KUKA KRL program: Machining1.src

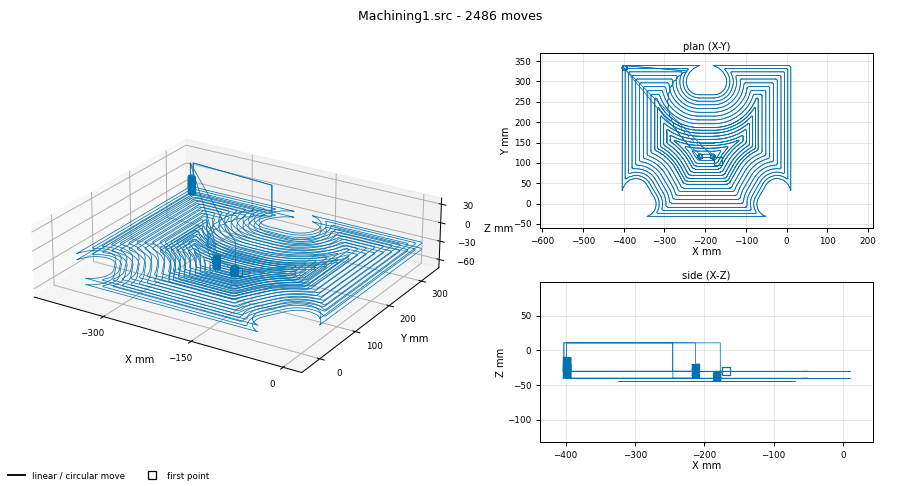
[picture p0: tool path of Machining1.src, 2486 of 2486 moves have a stored position in this frame; points joined in program order, loops and branches not executed]
&ACCESS RVP
&REL 1
&PARAM TEMPLATE = C:\KRC\Roboter\Template\vorgabe
&PARAM EDITMASK = *
DEF Machining1 ( )

; External program calls:
EXT Machining2()

CIRC {X -171.302,Y 100.492,Z -30.000,A 0.015,B 0.000,C 180.000},{X -168.190,Y 103.602,Z -30.000,A 0.015,B 0.000,C 180.000} C_DIS
CIRC {X -167.107,Y 105.546,Z -30.000,A 0.015,B 0.000,C -180.000},{X -166.084,Y 107.524,Z -30.000,A 0.015,B -0.000,C -180.000} C_DIS
CIRC {X -165.062,Y 109.501,Z -30.000,A 0.015,B 0.000,C -180.000},{X -163.978,Y 111.446,Z -30.000,A 0.015,B 0.000,C 180.000} C_DIS
CIRC {X -159.665,Y 118.376,Z -30.000,A 0.015,B 0.000,C 180.000},{X -154.910,Y 125.010,Z -30.000,A 0.015,B -0.000,C -180.000} C_DIS
CIRC {X -149.826,Y 131.393,Z -30.000,A 0.015,B 0.000,C 180.000},{X -144.514,Y 137.587,Z -30.000,A 0.015,B -0.000,C 180.000} C_DIS
CIRC {X -144.313,Y 139.468,Z -30.000,A 0.015,B 0.000,C 180.000},{X -146.029,Y 140.268,Z -30.000,A 0.015,B -0.000,C -180.000} C_DIS
CIRC {X -149.975,Y 139.497,Z -30.000,A 0.015,B 0.000,C -180.000},{X -153.909,Y 138.663,Z -30.000,A 0.015,B 0.000,C 180.000} C_DIS
CIRC {X -157.855,Y 137.887,Z -30.000,A 0.015,B 0.000,C 180.000},{X -161.833,Y 137.294,Z -30.000,A 0.015,B 0.000,C 180.000} C_DIS
CIRC {X -170.208,Y 136.495,Z -30.000,A 0.015,B 0.000,C -180.000},{X -178.617,Y 136.202,Z -30.000,A 0.015,B 0.000,C -180.000} C_DIS
LIN {X -214.895,Y 136.202,Z -30.000,A 0.015,B 0.000,C 180.000} C_DIS
CIRC {X -223.102,Y 136.522,Z -30.000,A 0.015,B 0.000,C 180.000},{X -231.259,Y 137.480,Z -30.000,A 0.015,B 0.000,C 180.000} C_DIS
CIRC {X -232.124,Y 137.616,Z -30.000,A 0.015,B 0.000,C -180.000},{X -232.988,Y 137.754,Z -30.000,A 0.015,B 0.000,C 180.000} C_DIS
CIRC {X -235.696,Y 139.055,Z -30.000,A 0.015,B -0.000,C 180.000},{X -237.254,Y 141.623,Z -30.000,A 0.015,B 0.000,C 180.000} C_DIS
CIRC {X -238.790,Y 144.198,Z -30.000,A 0.015,B 0.000,C 180.000},{X -241.463,Y 145.555,Z -30.000,A 0.015,B 0.000,C 180.000} C_DIS
CIRC {X -243.440,Y 145.946,Z -30.000,A 0.015,B -0.000,C 180.000},{X -245.411,Y 146.366,Z -30.000,A 0.015,B 0.000,C -180.000} C_DIS
CIRC {X -260.252,Y 150.338,Z -30.000,A 0.015,B 0.000,C 180.000},{X -274.679,Y 155.621,Z -30.000,A 0.015,B 0.000,C -180.000} C_DIS
CIRC {X -276.235,Y 155.093,Z -30.000,A 0.015,B -0.000,C -180.000},{X -275.907,Y 153.483,Z -30.000,A 0.015,B 0.000,C -180.000} C_DIS
CIRC {X -266.896,Y 146.130,Z -30.000,A 0.015,B -0.000,C -180.000},{X -258.464,Y 138.119,Z -30.000,A 0.015,B 0.000,C -180.000} C_DIS
CIRC {X -250.617,Y 129.537,Z -30.000,A 0.015,B 0.000,C 180.000},{X -243.351,Y 120.458,Z -30.000,A 0.015,B -0.000,C 180.000} C_DIS
CIRC {X -241.131,Y 117.362,Z -30.000,A 0.015,B 0.000,C -180.000},{X -239.037,Y 114.180,Z -30.000,A 0.015,B 0.000,C 180.000} C_DIS
CIRC {X -237.039,Y 110.937,Z -30.000,A 0.015,B -0.000,C -180.000},{X -235.105,Y 107.656,Z -30.000,A 0.015,B 0.000,C 180.000} C_DIS
CIRC {X -233.604,Y 104.954,Z -30.000,A 0.015,B 0.000,C 180.000},{X -232.188,Y 102.206,Z -30.000,A 0.015,B 0.000,C 180.000} C_DIS
CIRC {X -230.772,Y 99.459,Z -30.000,A 0.015,B 0.000,C -180.000},{X -229.270,Y 96.757,Z -30.000,A 0.015,B 0.000,C -180.000} C_DIS
CIRC {X -226.165,Y 93.648,Z -30.000,A 0.015,B 0.000,C 180.000},{X -221.922,Y 92.510,Z -30.000,A 0.015,B 0.000,C 180.000} C_DIS
LIN {X -171.602,Y 92.510,Z -30.000,A 0.015,B 0.000,C -180.000} C_DIS
CIRC {X -167.353,Y 93.648,Z -30.000,A 0.015,B 0.000,C -180.000},{X -164.241,Y 96.758,Z -30.000,A 0.015,B 0.000,C 180.000} C_DIS
CIRC {X -162.677,Y 99.566,Z -30.000,A 0.015,B 0.000,C 180.000},{X -161.200,Y 102.421,Z -30.000,A 0.015,B -0.000,C 180.000} C_DIS
CIRC {X -159.724,Y 105.276,Z -30.000,A 0.015,B 0.000,C 180.000},{X -158.160,Y 108.083,Z -30.000,A 0.015,B 0.000,C -180.000} C_DIS
CIRC {X -149.792,Y 120.931,Z -30.000,A 0.015,B -0.000,C -180.000},{X -140.107,Y 132.817,Z -30.000,A 0.015,B -0.000,C -180.000} C_DIS
CIRC {X -129.299,Y 143.685,Z -30.000,A 0.015,B 0.000,C -180.000},{X -117.547,Y 153.523,Z -30.000,A 0.015,B -0.000,C 180.000} C_DIS
CIRC {X -117.226,Y 155.134,Z -30.000,A 0.015,B 0.000,C 180.000},{X -118.785,Y 155.652,Z -30.000,A 0.015,B 0.000,C 180.000} C_DIS
CIRC {X -129.422,Y 151.590,Z -30.000,A 0.015,B 0.000,C -180.000},{X -140.331,Y 148.327,Z -30.000,A 0.015,B 0.000,C 180.000} C_DIS
CIRC {X -151.437,Y 145.826,Z -30.000,A 0.015,B -0.000,C -180.000},{X -162.682,Y 144.043,Z -30.000,A 0.015,B 0.000,C 180.000} C_DIS
CIRC {X -170.633,Y 143.295,Z -30.000,A 0.015,B 0.000,C 180.000},{X -178.617,Y 143.045,Z -30.000,A 0.015,B 0.000,C 180.000} C_DIS
LIN {X -214.895,Y 143.045,Z -30.000,A 0.015,B 0.000,C 180.000} C_DIS
CIRC {X -228.238,Y 143.674,Z -30.000,A 0.015,B 0.000,C 180.000},{X -241.463,Y 145.555,Z -30.000,A 0.015,B 0.000,C -180.000} C_DIS
CIRC {X -244.234,Y 147.015,Z -30.000,A 0.015,B 0.000,C 180.000},{X -245.715,Y 149.775,Z -30.000,A 0.015,B 0.000,C -180.000} C_DIS
CIRC {X -247.142,Y 152.546,Z -30.000,A 0.015,B 0.000,C -180.000},{X -249.821,Y 154.137,Z -30.000,A 0.015,B -0.000,C -180.000} C_DIS
LIN {X -250.098,Y 154.210,Z -30.000,A 0.015,B -0.000,C -180.000} C_DIS
CIRC {X -267.011,Y 159.678,Z -30.000,A 0.015,B 0.000,C -180.000},{X -283.228,Y 166.955,Z -30.000,A 0.015,B 0.000,C 180.000} C_DIS
CIRC {X -285.491,Y 166.874,Z -30.000,A 0.015,B 0.000,C -180.000},{X -286.600,Y 164.900,Z -30.000,A 0.015,B 0.000,C 180.000} C_DIS
LIN {X -286.600,Y 156.568,Z -30.000,A 0.015,B 0.000,C 180.000} C_DIS
CIRC {X -285.833,Y 153.428,Z -30.000,A 0.015,B 0.000,C 180.000},{X -283.705,Y 150.996,Z -30.000,A 0.015,B 0.000,C 180.000} C_DIS
CIRC {X -271.141,Y 141.152,Z -30.000,A 0.015,B 0.000,C -180.000},{X -259.666,Y 130.058,Z -30.000,A 0.015,B 0.000,C -180.000} C_DIS
CIRC {X -249.460,Y 117.780,Z -30.000,A 0.015,B 0.000,C 180.000},{X -240.715,Y 104.423,Z -30.000,A 0.015,B 0.000,C -180.000} C_DIS
CIRC {X -238.751,Y 100.888,Z -30.000,A 0.015,B 0.000,C 180.000},{X -236.898,Y 97.293,Z -30.000,A 0.015,B 0.000,C -180.000} C_DIS
CIRC {X -235.045,Y 93.698,Z -30.000,A 0.015,B -0.000,C -180.000},{X -233.081,Y 90.163,Z -30.000,A 0.015,B -0.000,C -180.000} C_DIS
CIRC {X -229.976,Y 87.054,Z -30.000,A 0.015,B 0.000,C 180.000},{X -225.732,Y 85.916,Z -30.000,A 0.015,B 0.000,C 180.000} C_DIS
LIN {X -167.797,Y 85.916,Z -30.000,A 0.015,B 0.000,C 180.000} C_DIS
CIRC {X -163.547,Y 87.055,Z -30.000,A 0.015,B -0.000,C 180.000},{X -160.436,Y 90.164,Z -30.000,A 0.015,B 0.000,C 180.000} C_DIS
CIRC {X -158.408,Y 93.803,Z -30.000,A 0.015,B 0.000,C -180.000},{X -156.495,Y 97.504,Z -30.000,A 0.015,B 0.000,C -180.000} C_DIS
CIRC {X -154.582,Y 101.205,Z -30.000,A 0.015,B 0.000,C 180.000},{X -152.554,Y 104.844,Z -30.000,A 0.015,B 0.000,C -180.000} C_DIS
CIRC {X -143.851,Y 118.092,Z -30.000,A 0.015,B 0.000,C 180.000},{X -133.694,Y 130.260,Z -30.000,A 0.015,B 0.000,C 180.000} C_DIS
CIRC {X -122.283,Y 141.253,Z -30.000,A 0.015,B 0.000,C 180.000},{X -109.806,Y 151.020,Z -30.000,A 0.015,B -0.000,C -180.000} C_DIS
CIRC {X -107.679,Y 153.453,Z -30.000,A 0.015,B 0.000,C 180.000},{X -106.912,Y 156.592,Z -30.000,A 0.015,B 0.000,C -180.000} C_DIS
LIN {X -106.913,Y 164.900,Z -30.000,A 0.015,B -0.000,C 180.000} C_DIS
CIRC {X -108.021,Y 166.866,Z -30.000,A 0.015,B 0.000,C -180.000},{X -110.278,Y 166.935,Z -30.000,A 0.015,B 0.000,C 180.000} C_DIS
CIRC {X -122.965,Y 161.035,Z -30.000,A 0.015,B 0.000,C 180.000},{X -136.157,Y 156.372,Z -30.000,A 0.015,B -0.000,C -180.000} C_DIS
CIRC {X -149.710,Y 152.908,Z -30.000,A 0.015,B -0.000,C -180.000},{X -163.504,Y 150.586,Z -30.000,A 0.015,B -0.000,C -180.000} C_DIS
CIRC {X -171.046,Y 149.876,Z -30.000,A 0.015,B 0.000,C 180.000},{X -178.617,Y 149.639,Z -30.000,A 0.015,B 0.000,C 180.000} C_DIS
LIN {X -214.895,Y 149.639,Z -30.000,A 0.015,B 0.000,C -180.000} C_DIS
CIRC {X -232.503,Y 150.768,Z -30.000,A 0.015,B -0.000,C 180.000},{X -249.821,Y 154.137,Z -30.000,A 0.015,B -0.000,C 180.000} C_DIS
CIRC {X -253.023,Y 156.105,Z -30.000,A 0.015,B 0.000,C -180.000},{X -254.587,Y 159.522,Z -30.000,A 0.015,B 0.000,C -180.000} C_DIS
CIRC {X -256.087,Y 162.948,Z -30.000,A 0.015,B 0.000,C 180.000},{X -259.170,Y 165.064,Z -30.000,A 0.015,B 0.000,C 180.000} C_DIS
CIRC {X -269.017,Y 168.755,Z -30.000,A 0.015,B 0.000,C -180.000},{X -278.578,Y 173.132,Z -30.000,A 0.015,B 0.000,C -180.000} C_DIS
CIRC {X -281.907,Y 174.946,Z -30.000,A 0.015,B 0.000,C -180.000},{X -285.103,Y 176.984,Z -30.000,A 0.015,B 0.000,C 180.000} C_DIS
CIRC {X -288.241,Y 179.109,Z -30.000,A 0.015,B 0.000,C 180.000},{X -291.406,Y 181.191,Z -30.000,A 0.015,B 0.000,C 180.000} C_DIS
CIRC {X -293.577,Y 181.275,Z -30.000,A 0.015,B 0.000,C 180.000},{X -294.687,Y 179.408,Z -30.000,A 0.015,B 0.000,C 180.000} C_DIS
LIN {X -294.686,Y 153.798,Z -30.000,A 0.015,B 0.000,C 180.000} C_DIS
CIRC {X -293.590,Y 149.349,Z -30.000,A 0.015,B 0.000,C 180.000},{X -290.552,Y 145.919,Z -30.000,A 0.015,B 0.000,C 180.000} C_DIS
CIRC {X -271.422,Y 130.249,Z -30.000,A 0.015,B 0.000,C -180.000},{X -255.107,Y 111.666,Z -30.000,A 0.015,B 0.000,C 180.000} C_DIS
CIRC {X -251.230,Y 106.146,Z -30.000,A 0.015,B 0.000,C 180.000},{X -247.689,Y 100.404,Z -30.000,A 0.015,B -0.000,C 180.000} C_DIS
CIRC {X -245.145,Y 95.855,Z -30.000,A 0.015,B -0.000,C 180.000},{X -242.722,Y 91.240,Z -30.000,A 0.015,B 0.000,C 180.000} C_DIS
CIRC {X -240.298,Y 86.626,Z -30.000,A 0.015,B 0.000,C 180.000},{X -237.754,Y 82.077,Z -30.000,A 0.015,B 0.000,C -180.000} C_DIS
CIRC {X -234.649,Y 78.968,Z -30.000,A 0.015,B 0.000,C 180.000},{X -230.405,Y 77.830,Z -30.000,A 0.015,B 0.000,C -180.000} C_DIS
LIN {X -163.130,Y 77.830,Z -30.000,A 0.015,B 0.000,C 180.000} C_DIS
CIRC {X -158.881,Y 78.968,Z -30.000,A 0.015,B -0.000,C 180.000},{X -155.769,Y 82.077,Z -30.000,A 0.015,B 0.000,C 180.000} C_DIS
CIRC {X -153.160,Y 86.728,Z -30.000,A 0.015,B 0.000,C 180.000},{X -150.670,Y 91.443,Z -30.000,A 0.015,B 0.000,C 180.000} C_DIS
CIRC {X -148.181,Y 96.158,Z -30.000,A 0.015,B -0.000,C 180.000},{X -145.572,Y 100.809,Z -30.000,A 0.015,B 0.000,C -180.000} C_DIS
CIRC {X -136.969,Y 113.835,Z -30.000,A 0.015,B 0.000,C 180.000},{X -126.877,Y 125.745,Z -30.000,A 0.015,B -0.000,C -180.000} C_DIS
CIRC {X -115.507,Y 136.435,Z -30.000,A 0.015,B 0.000,C 180.000},{X -103.058,Y 145.845,Z -30.000,A 0.015,B 0.000,C -180.000} C_DIS
CIRC {X -99.949,Y 149.299,Z -30.000,A 0.015,B 0.000,C 180.000},{X -98.826,Y 153.807,Z -30.000,A 0.015,B 0.000,C 180.000} C_DIS
LIN {X -98.826,Y 179.417,Z -30.000,A 0.015,B 0.000,C -180.000} C_DIS
CIRC {X -99.933,Y 181.277,Z -30.000,A 0.015,B -0.000,C -180.000},{X -102.095,Y 181.192,Z -30.000,A 0.015,B 0.000,C -180.000} C_DIS
CIRC {X -110.083,Y 176.279,Z -30.000,A 0.015,B 0.000,C 180.000},{X -118.304,Y 171.770,Z -30.000,A 0.015,B -0.000,C -180.000} C_DIS
CIRC {X -126.806,Y 167.804,Z -30.000,A 0.015,B 0.000,C 180.000},{X -135.601,Y 164.537,Z -30.000,A 0.015,B 0.000,C 180.000} C_DIS
CIRC {X -155.043,Y 159.783,Z -30.000,A 0.015,B -0.000,C -180.000},{X -174.979,Y 158.001,Z -30.000,A 0.015,B 0.000,C 180.000} C_DIS
LIN {X -214.895,Y 157.726,Z -30.000,A 0.015,B -0.000,C -180.000} C_DIS
CIRC {X -231.386,Y 158.726,Z -30.000,A 0.015,B 0.000,C 180.000},{X -247.636,Y 161.713,Z -30.000,A 0.015,B 0.000,C -180.000} C_DIS
CIRC {X -253.437,Y 163.272,Z -30.000,A 0.015,B 0.000,C 180.000},{X -259.170,Y 165.064,Z -30.000,A 0.015,B -0.000,C -180.000} C_DIS
CIRC {X -262.205,Y 167.235,Z -30.000,A 0.015,B 0.000,C 180.000},{X -263.500,Y 170.734,Z -30.000,A 0.015,B 0.000,C -180.000} C_DIS
CIRC {X -264.716,Y 174.238,Z -30.000,A 0.015,B 0.000,C 180.000},{X -267.594,Y 176.578,Z -30.000,A 0.015,B -0.000,C 180.000} C_DIS
CIRC {X -271.373,Y 178.266,Z -30.000,A 0.015,B 0.000,C 180.000},{X -275.101,Y 180.067,Z -30.000,A 0.015,B 0.000,C 180.000} C_DIS
CIRC {X -281.532,Y 183.634,Z -30.000,A 0.015,B 0.000,C -180.000},{X -287.644,Y 187.725,Z -30.000,A 0.015,B 0.000,C 180.000} C_DIS
CIRC {X -293.535,Y 192.117,Z -30.000,A 0.015,B -0.000,C -180.000},{X -299.344,Y 196.618,Z -30.000,A 0.015,B 0.000,C -180.000} C_DIS
CIRC {X -301.411,Y 196.843,Z -30.000,A 0.015,B -0.000,C 180.000},{X -302.515,Y 195.081,Z -30.000,A 0.015,B 0.000,C 180.000} C_DIS
LIN {X -302.514,Y 149.210,Z -30.000,A 0.015,B 0.000,C -180.000} C_DIS
CIRC {X -301.418,Y 144.941,Z -30.000,A 0.015,B 0.000,C -180.000},{X -298.400,Y 141.729,Z -30.000,A 0.015,B 0.000,C 180.000} C_DIS
CIRC {X -287.970,Y 134.375,Z -30.000,A 0.015,B 0.000,C 180.000},{X -278.306,Y 126.039,Z -30.000,A 0.015,B 0.000,C 180.000} C_DIS
CIRC {X -269.440,Y 116.864,Z -30.000,A 0.015,B 0.000,C -180.000},{X -261.376,Y 106.977,Z -30.000,A 0.015,B 0.000,C 180.000} C_DIS
CIRC {X -257.767,Y 101.839,Z -30.000,A 0.015,B 0.000,C 180.000},{X -254.471,Y 96.496,Z -30.000,A 0.015,B 0.000,C 180.000} C_DIS
CIRC {X -251.364,Y 90.966,Z -30.000,A 0.015,B -0.000,C -180.000},{X -248.375,Y 85.372,Z -30.000,A 0.015,B -0.000,C 180.000} C_DIS
CIRC {X -245.386,Y 79.778,Z -30.000,A 0.015,B 0.000,C -180.000},{X -242.278,Y 74.249,Z -30.000,A 0.015,B -0.000,C -180.000} C_DIS
CIRC {X -239.173,Y 71.140,Z -30.000,A 0.015,B 0.000,C 180.000},{X -234.929,Y 70.002,Z -30.000,A 0.015,B 0.000,C 180.000} C_DIS
LIN {X -158.613,Y 70.002,Z -30.000,A 0.015,B 0.000,C 180.000} C_DIS
CIRC {X -154.364,Y 71.140,Z -30.000,A 0.015,B 0.000,C 180.000},{X -151.252,Y 74.249,Z -30.000,A 0.015,B 0.000,C -180.000} C_DIS
LIN {X -138.794,Y 96.892,Z -30.000,A 0.015,B 0.000,C -180.000} C_DIS
CIRC {X -130.024,Y 110.028,Z -30.000,A 0.015,B 0.000,C 180.000},{X -119.634,Y 121.923,Z -30.000,A 0.015,B 0.000,C -180.000} C_DIS
CIRC {X -107.912,Y 132.494,Z -30.000,A 0.015,B -0.000,C 180.000},{X -95.112,Y 141.730,Z -30.000,A 0.015,B 0.000,C 180.000} C_DIS
CIRC {X -92.093,Y 144.970,Z -30.000,A 0.015,B 0.000,C 180.000},{X -90.997,Y 149.261,Z -30.000,A 0.015,B 0.000,C -180.000} C_DIS
LIN {X -90.999,Y 195.079,Z -30.000,A 0.015,B 0.000,C 180.000} C_DIS
CIRC {X -92.103,Y 196.841,Z -30.000,A 0.015,B -0.000,C 180.000},{X -94.171,Y 196.616,Z -30.000,A 0.015,B 0.000,C -180.000} C_DIS
CIRC {X -104.346,Y 189.131,Z -30.000,A 0.015,B 0.000,C 180.000},{X -115.009,Y 182.357,Z -30.000,A 0.015,B 0.000,C -180.000} C_DIS
CIRC {X -126.237,Y 176.544,Z -30.000,A 0.015,B -0.000,C 180.000},{X -138.028,Y 171.980,Z -30.000,A 0.015,B 0.000,C -180.000} C_DIS
CIRC {X -156.878,Y 167.393,Z -30.000,A 0.015,B 0.000,C -180.000},{X -176.208,Y 165.732,Z -30.000,A 0.015,B 0.000,C 180.000} C_DIS
LIN {X -214.895,Y 165.554,Z -30.000,A 0.015,B 0.000,C 180.000} C_DIS
CIRC {X -230.483,Y 166.493,Z -30.000,A 0.015,B 0.000,C 180.000},{X -245.845,Y 169.297,Z -30.000,A 0.015,B 0.000,C -180.000} C_DIS
CIRC {X -256.869,Y 172.489,Z -30.000,A 0.015,B -0.000,C 180.000},{X -267.594,Y 176.578,Z -30.000,A 0.015,B 0.000,C 180.000} C_DIS
CIRC {X -270.381,Y 178.951,Z -30.000,A 0.015,B 0.000,C 180.000},{X -271.340,Y 182.484,Z -30.000,A 0.015,B 0.000,C 180.000} C_DIS
CIRC {X -272.205,Y 186.013,Z -30.000,A 0.015,B 0.000,C 180.000},{X -274.787,Y 188.568,Z -30.000,A 0.015,B -0.000,C -180.000} C_DIS
CIRC {X -292.023,Y 200.077,Z -30.000,A 0.015,B -0.000,C -180.000},{X -307.098,Y 214.300,Z -30.000,A 0.015,B 0.000,C 180.000} C_DIS
CIRC {X -308.980,Y 214.762,Z -30.000,A 0.015,B -0.000,C 180.000},{X -310.080,Y 213.167,Z -30.000,A 0.015,B -0.000,C -180.000} C_DIS
LIN {X -310.079,Y 144.563,Z -30.000,A 0.015,B 0.000,C 180.000} C_DIS
CIRC {X -308.981,Y 140.472,Z -30.000,A 0.015,B 0.000,C -180.000},{X -305.984,Y 137.478,Z -30.000,A 0.015,B 0.000,C -180.000} C_DIS
CIRC {X -295.014,Y 130.299,Z -30.000,A 0.015,B 0.000,C 180.000},{X -284.926,Y 121.925,Z -30.000,A 0.015,B -0.000,C -180.000} C_DIS
CIRC {X -275.743,Y 112.578,Z -30.000,A 0.015,B -0.000,C -180.000},{X -267.433,Y 102.447,Z -30.000,A 0.015,B 0.000,C -180.000} C_DIS
CIRC {X -264.084,Y 97.678,Z -30.000,A 0.015,B 0.000,C 180.000},{X -261.025,Y 92.719,Z -30.000,A 0.015,B 0.000,C 180.000} C_DIS
LIN {X -246.650,Y 66.684,Z -30.000,A 0.015,B 0.000,C -180.000} C_DIS
CIRC {X -243.545,Y 63.575,Z -30.000,A 0.015,B 0.000,C -180.000},{X -239.301,Y 62.437,Z -30.000,A 0.015,B 0.000,C 180.000} C_DIS
LIN {X -154.248,Y 62.437,Z -30.000,A 0.015,B 0.000,C -180.000} C_DIS
CIRC {X -149.998,Y 63.575,Z -30.000,A 0.015,B 0.000,C 180.000},{X -146.887,Y 66.685,Z -30.000,A 0.015,B 0.000,C 180.000} C_DIS
LIN {X -132.244,Y 93.107,Z -30.000,A 0.015,B 0.000,C 180.000} C_DIS
CIRC {X -123.362,Y 106.324,Z -30.000,A 0.015,B 0.000,C -180.000},{X -112.778,Y 118.222,Z -30.000,A 0.015,B 0.000,C 180.000} C_DIS
CIRC {X -100.749,Y 128.648,Z -30.000,A 0.015,B 0.000,C -180.000},{X -87.524,Y 137.509,Z -30.000,A 0.015,B 0.000,C -180.000} C_DIS
CIRC {X -84.528,Y 140.526,Z -30.000,A 0.015,B -0.000,C 180.000},{X -83.433,Y 144.635,Z -30.000,A 0.015,B 0.000,C -180.000} C_DIS
LIN {X -83.435,Y 213.163,Z -30.000,A 0.015,B 0.000,C -180.000} C_DIS
CIRC {X -84.535,Y 214.758,Z -30.000,A 0.015,B 0.000,C -180.000},{X -86.417,Y 214.296,Z -30.000,A 0.015,B 0.000,C 180.000} C_DIS
CIRC {X -103.225,Y 198.757,Z -30.000,A 0.015,B 0.000,C -180.000},{X -122.750,Y 186.812,Z -30.000,A 0.015,B 0.000,C 180.000} C_DIS
CIRC {X -144.065,Y 178.566,Z -30.000,A 0.015,B -0.000,C 180.000},{X -166.434,Y 173.881,Z -30.000,A 0.015,B 0.000,C 180.000} C_DIS
LIN {X -214.895,Y 173.118,Z -30.000,A 0.015,B -0.000,C 180.000} C_DIS
CIRC {X -245.822,Y 177.043,Z -30.000,A 0.015,B 0.000,C 180.000},{X -274.787,Y 188.568,Z -30.000,A 0.015,B 0.000,C 180.000} C_DIS
CIRC {X -277.258,Y 191.114,Z -30.000,A 0.015,B 0.000,C 180.000},{X -277.893,Y 194.605,Z -30.000,A 0.015,B 0.000,C -180.000} C_DIS
CIRC {X -278.464,Y 198.089,Z -30.000,A 0.015,B -0.000,C 180.000},{X -280.787,Y 200.746,Z -30.000,A 0.015,B -0.000,C -180.000} C_DIS
CIRC {X -284.969,Y 203.559,Z -30.000,A 0.015,B 0.000,C -180.000},{X -289.045,Y 206.523,Z -30.000,A 0.015,B 0.000,C -180.000} C_DIS
CIRC {X -296.399,Y 212.790,Z -30.000,A 0.015,B 0.000,C -180.000},{X -302.966,Y 219.879,Z -30.000,A 0.015,B 0.000,C 180.000} C_DIS
CIRC {X -308.886,Y 227.498,Z -30.000,A 0.015,B -0.000,C -180.000},{X -314.377,Y 235.434,Z -30.000,A 0.015,B -0.000,C -180.000} C_DIS
CIRC {X -316.098,Y 236.067,Z -30.000,A 0.015,B 0.000,C 180.000},{X -317.194,Y 234.597,Z -30.000,A 0.015,B 0.000,C 180.000} C_DIS
LIN {X -317.192,Y 140.213,Z -30.000,A 0.015,B 0.000,C 180.000} C_DIS
CIRC {X -316.058,Y 136.125,Z -30.000,A 0.015,B 0.000,C -180.000},{X -312.979,Y 133.205,Z -30.000,A 0.015,B 0.000,C -180.000} C_DIS
CIRC {X -292.253,Y 119.088,Z -30.000,A 0.015,B 0.000,C -180.000},{X -275.088,Y 100.805,Z -30.000,A 0.015,B -0.000,C 180.000} C_DIS
CIRC {X -273.004,Y 97.971,Z -30.000,A 0.015,B 0.000,C -180.000},{X -270.965,Y 95.104,Z -30.000,A 0.015,B 0.000,C 180.000} C_DIS
CIRC {X -269.012,Y 92.177,Z -30.000,A 0.015,B 0.000,C 180.000},{X -267.189,Y 89.167,Z -30.000,A 0.015,B 0.000,C 180.000} C_DIS
LIN {X -250.742,Y 59.538,Z -30.000,A 0.015,B 0.000,C 180.000} C_DIS
CIRC {X -247.660,Y 56.453,Z -30.000,A 0.015,B 0.000,C 180.000},{X -243.449,Y 55.324,Z -30.000,A 0.015,B -0.000,C -180.000} C_DIS
LIN {X -150.080,Y 55.324,Z -30.000,A 0.015,B 0.000,C -180.000} C_DIS
CIRC {X -145.885,Y 56.447,Z -30.000,A 0.015,B -0.000,C 180.000},{X -142.813,Y 59.517,Z -30.000,A 0.015,B 0.000,C 180.000} C_DIS
LIN {X -126.086,Y 89.548,Z -30.000,A 0.015,B 0.000,C 180.000} C_DIS
CIRC {X -106.380,Y 114.666,Z -30.000,A 0.015,B 0.000,C -180.000},{X -80.454,Y 133.297,Z -30.000,A 0.015,B 0.000,C -180.000} C_DIS
CIRC {X -77.433,Y 136.144,Z -30.000,A 0.015,B 0.000,C 180.000},{X -76.319,Y 140.143,Z -30.000,A 0.015,B 0.000,C -180.000} C_DIS
LIN {X -76.322,Y 234.602,Z -30.000,A 0.015,B 0.000,C 180.000} C_DIS
CIRC {X -77.419,Y 236.069,Z -30.000,A 0.015,B 0.000,C 180.000},{X -79.136,Y 235.433,Z -30.000,A 0.015,B 0.000,C -180.000} C_DIS
CIRC {X -85.589,Y 226.331,Z -30.000,A 0.015,B 0.000,C -180.000},{X -92.790,Y 217.807,Z -30.000,A 0.015,B -0.000,C 180.000} C_DIS
CIRC {X -100.722,Y 209.957,Z -30.000,A 0.015,B 0.000,C 180.000},{X -109.355,Y 202.884,Z -30.000,A 0.015,B 0.000,C 180.000} C_DIS
CIRC {X -120.709,Y 195.513,Z -30.000,A 0.015,B -0.000,C 180.000},{X -132.910,Y 189.647,Z -30.000,A 0.015,B 0.000,C -180.000} C_DIS
CIRC {X -145.694,Y 185.225,Z -30.000,A 0.015,B 0.000,C 180.000},{X -158.864,Y 182.136,Z -30.000,A 0.015,B -0.000,C -180.000} C_DIS
CIRC {X -172.795,Y 180.330,Z -30.000,A 0.015,B 0.000,C -180.000},{X -186.837,Y 179.928,Z -30.000,A 0.015,B -0.000,C 180.000} C_DIS
LIN {X -214.895,Y 180.232,Z -30.000,A 0.015,B 0.000,C -180.000} C_DIS
CIRC {X -234.824,Y 182.020,Z -30.000,A 0.015,B 0.000,C -180.000},{X -254.115,Y 187.329,Z -30.000,A 0.015,B 0.000,C 180.000} C_DIS
CIRC {X -267.814,Y 193.316,Z -30.000,A 0.015,B 0.000,C -180.000},{X -280.787,Y 200.746,Z -30.000,A 0.015,B 0.000,C 180.000} C_DIS
CIRC {X -282.747,Y 203.101,Z -30.000,A 0.015,B 0.000,C 180.000},{X -283.016,Y 206.154,Z -30.000,A 0.015,B 0.000,C -180.000} C_DIS
CIRC {X -283.201,Y 209.188,Z -30.000,A 0.015,B -0.000,C -180.000},{X -284.951,Y 211.674,Z -30.000,A 0.015,B 0.000,C 180.000} C_DIS
CIRC {X -304.568,Y 232.271,Z -30.000,A 0.015,B 0.000,C 180.000},{X -318.317,Y 257.172,Z -30.000,A 0.015,B 0.000,C -180.000} C_DIS
CIRC {X -321.488,Y 258.916,Z -30.000,A 0.015,B 0.000,C 180.000},{X -323.796,Y 256.128,Z -30.000,A 0.015,B 0.000,C 180.000} C_DIS
LIN {X -323.792,Y 135.950,Z -30.000,A 0.015,B 0.000,C -180.000} C_DIS
CIRC {X -322.699,Y 132.062,Z -30.000,A 0.015,B 0.000,C -180.000},{X -319.740,Y 129.313,Z -30.000,A 0.015,B 0.000,C -180.000} C_DIS
CIRC {X -312.688,Y 125.465,Z -30.000,A 0.015,B 0.000,C 180.000},{X -305.836,Y 121.270,Z -30.000,A 0.015,B 0.000,C 180.000} C_DIS
CIRC {X -299.286,Y 116.609,Z -30.000,A 0.015,B 0.000,C -180.000},{X -293.174,Y 111.386,Z -30.000,A 0.015,B 0.000,C -180.000} C_DIS
CIRC {X -281.197,Y 98.287,Z -30.000,A 0.015,B 0.000,C 180.000},{X -271.423,Y 83.470,Z -30.000,A 0.015,B 0.000,C 180.000} C_DIS
LIN {X -254.485,Y 52.785,Z -30.000,A 0.015,B 0.000,C 180.000} C_DIS
CIRC {X -251.598,Y 49.814,Z -30.000,A 0.015,B 0.000,C -180.000},{X -247.603,Y 48.723,Z -30.000,A 0.015,B 0.000,C 180.000} C_DIS
LIN {X -145.892,Y 48.723,Z -30.000,A 0.015,B 0.000,C -180.000} C_DIS
CIRC {X -141.915,Y 49.815,Z -30.000,A 0.015,B 0.000,C 180.000},{X -139.052,Y 52.783,Z -30.000,A 0.015,B -0.000,C 180.000} C_DIS
LIN {X -119.937,Y 86.451,Z -30.000,A 0.015,B 0.000,C -180.000} C_DIS
CIRC {X -108.721,Y 102.309,Z -30.000,A 0.015,B 0.000,C 180.000},{X -95.059,Y 116.117,Z -30.000,A 0.015,B 0.000,C -180.000} C_DIS
CIRC {X -90.117,Y 119.963,Z -30.000,A 0.015,B 0.000,C 180.000},{X -84.834,Y 123.328,Z -30.000,A 0.015,B 0.000,C 180.000} C_DIS
CIRC {X -79.366,Y 126.369,Z -30.000,A 0.015,B 0.000,C 180.000},{X -73.823,Y 129.272,Z -30.000,A 0.015,B -0.000,C -180.000} C_DIS
CIRC {X -70.827,Y 132.038,Z -30.000,A 0.015,B -0.000,C 180.000},{X -69.719,Y 135.963,Z -30.000,A 0.015,B 0.000,C -180.000} C_DIS
LIN {X -69.722,Y 256.114,Z -30.000,A 0.015,B 0.000,C 180.000} C_DIS
CIRC {X -72.029,Y 258.902,Z -30.000,A 0.015,B -0.000,C 180.000},{X -75.200,Y 257.158,Z -30.000,A 0.015,B 0.000,C 180.000} C_DIS
CIRC {X -88.997,Y 232.325,Z -30.000,A 0.015,B 0.000,C 180.000},{X -108.733,Y 211.892,Z -30.000,A 0.015,B 0.000,C -180.000} C_DIS
CIRC {X -132.945,Y 197.083,Z -30.000,A 0.015,B 0.000,C -180.000},{X -160.040,Y 188.631,Z -30.000,A 0.015,B -0.000,C 180.000} C_DIS
CIRC {X -173.679,Y 186.871,Z -30.000,A 0.015,B 0.000,C 180.000},{X -187.427,Y 186.503,Z -30.000,A 0.015,B 0.000,C 180.000} C_DIS
LIN {X -214.895,Y 186.832,Z -30.000,A 0.015,B 0.000,C 180.000} C_DIS
CIRC {X -252.060,Y 193.226,Z -30.000,A 0.015,B 0.000,C 180.000},{X -284.951,Y 211.674,Z -30.000,A 0.015,B 0.000,C 180.000} C_DIS
CIRC {X -287.404,Y 215.341,Z -30.000,A 0.015,B 0.000,C 180.000},{X -287.362,Y 219.752,Z -30.000,A 0.015,B -0.000,C -180.000} C_DIS
CIRC {X -287.175,Y 224.118,Z -30.000,A 0.015,B 0.000,C 180.000},{X -289.230,Y 227.974,Z -30.000,A 0.015,B -0.000,C 180.000} C_DIS
CIRC {X -302.150,Y 245.093,Z -30.000,A 0.015,B 0.000,C -180.000},{X -311.057,Y 264.604,Z -30.000,A 0.015,B -0.000,C 180.000} C_DIS
CIRC {X -313.161,Y 267.478,Z -30.000,A 0.015,B 0.000,C -180.000},{X -316.550,Y 268.574,Z -30.000,A 0.015,B 0.000,C 180.000} C_DIS
LIN {X -329.306,Y 268.574,Z -30.000,A 0.015,B -0.000,C 180.000} C_DIS
CIRC {X -332.030,Y 267.446,Z -30.000,A 0.015,B 0.000,C 180.000},{X -333.159,Y 264.721,Z -30.000,A 0.015,B 0.000,C 180.000} C_DIS
LIN {X -333.155,Y 129.665,Z -30.000,A 0.015,B 0.000,C -180.000} C_DIS
CIRC {X -332.018,Y 125.864,Z -30.000,A 0.015,B -0.000,C -180.000},{X -328.982,Y 123.310,Z -30.000,A 0.015,B 0.000,C 180.000} C_DIS
CIRC {X -314.641,Y 115.756,Z -30.000,A 0.015,B 0.000,C 180.000},{X -301.608,Y 106.118,Z -30.000,A 0.015,B 0.000,C -180.000} C_DIS
CIRC {X -290.267,Y 94.523,Z -30.000,A 0.015,B 0.000,C -180.000},{X -281.020,Y 81.197,Z -30.000,A 0.015,B -0.000,C 180.000} C_DIS
LIN {X -263.166,Y 49.553,Z -30.000,A 0.015,B 0.000,C 180.000} C_DIS
CIRC {X -262.354,Y 48.051,Z -30.000,A 0.015,B -0.000,C -180.000},{X -261.624,Y 46.507,Z -30.000,A 0.015,B 0.000,C -180.000} C_DIS
CIRC {X -260.930,Y 44.947,Z -30.000,A 0.015,B -0.000,C 180.000},{X -260.224,Y 43.393,Z -30.000,A 0.015,B -0.000,C -180.000} C_DIS
CIRC {X -257.670,Y 40.455,Z -30.000,A 0.015,B -0.000,C -180.000},{X -253.933,Y 39.361,Z -30.000,A 0.015,B 0.000,C -180.000} C_DIS
LIN {X -139.560,Y 39.361,Z -30.000,A 0.015,B 0.000,C -180.000} C_DIS
CIRC {X -135.817,Y 40.463,Z -30.000,A 0.015,B 0.000,C 180.000},{X -133.267,Y 43.417,Z -30.000,A 0.015,B 0.000,C 180.000} C_DIS
CIRC {X -132.520,Y 45.080,Z -30.000,A 0.015,B 0.000,C 180.000},{X -131.783,Y 46.748,Z -30.000,A 0.015,B 0.000,C 180.000} C_DIS
CIRC {X -131.006,Y 48.398,Z -30.000,A 0.015,B 0.000,C -180.000},{X -130.137,Y 50.002,Z -30.000,A 0.015,B 0.000,C -180.000} C_DIS
LIN {X -112.264,Y 81.560,Z -30.000,A 0.015,B 0.000,C -180.000} C_DIS
CIRC {X -103.050,Y 94.803,Z -30.000,A 0.015,B -0.000,C 180.000},{X -91.754,Y 106.322,Z -30.000,A 0.015,B 0.000,C 180.000} C_DIS
CIRC {X -78.769,Y 115.880,Z -30.000,A 0.015,B 0.000,C 180.000},{X -64.475,Y 123.341,Z -30.000,A 0.015,B -0.000,C 180.000} C_DIS
CIRC {X -61.478,Y 125.844,Z -30.000,A 0.015,B 0.000,C 180.000},{X -60.356,Y 129.584,Z -30.000,A 0.015,B -0.000,C 180.000} C_DIS
LIN {X -60.359,Y 264.728,Z -30.000,A 0.015,B 0.000,C -180.000} C_DIS
CIRC {X -61.488,Y 267.452,Z -30.000,A 0.015,B 0.000,C 180.000},{X -64.213,Y 268.581,Z -30.000,A 0.015,B 0.000,C 180.000} C_DIS
LIN {X -76.960,Y 268.580,Z -30.000,A 0.015,B 0.000,C 180.000} C_DIS
CIRC {X -80.349,Y 267.484,Z -30.000,A 0.015,B 0.000,C -180.000},{X -82.453,Y 264.610,Z -30.000,A 0.015,B -0.000,C -180.000} C_DIS
CIRC {X -94.521,Y 240.300,Z -30.000,A 0.015,B 0.000,C -180.000},{X -112.907,Y 220.337,Z -30.000,A 0.015,B 0.000,C -180.000} C_DIS
CIRC {X -135.878,Y 205.990,Z -30.000,A 0.015,B 0.000,C 180.000},{X -161.708,Y 197.844,Z -30.000,A 0.015,B 0.000,C -180.000} C_DIS
CIRC {X -174.934,Y 196.149,Z -30.000,A 0.015,B 0.000,C 180.000},{X -188.265,Y 195.828,Z -30.000,A 0.015,B 0.000,C 180.000} C_DIS
CIRC {X -201.579,Y 196.103,Z -30.000,A 0.015,B 0.000,C 180.000},{X -214.895,Y 196.195,Z -30.000,A 0.015,B 0.000,C -180.000} C_DIS
CIRC {X -245.904,Y 200.967,Z -30.000,A 0.015,B 0.000,C 180.000},{X -274.043,Y 214.843,Z -30.000,A 0.015,B 0.000,C 180.000} C_DIS
CIRC {X -281.972,Y 221.020,Z -30.000,A 0.015,B -0.000,C 180.000},{X -289.230,Y 227.974,Z -30.000,A 0.015,B 0.000,C 180.000} C_DIS
CIRC {X -291.334,Y 232.250,Z -30.000,A 0.015,B -0.000,C -180.000},{X -290.673,Y 236.969,Z -30.000,A 0.015,B 0.000,C 180.000} C_DIS
CIRC {X -289.841,Y 241.609,Z -30.000,A 0.015,B 0.000,C -180.000},{X -291.428,Y 246.048,Z -30.000,A 0.015,B 0.000,C -180.000} C_DIS
CIRC {X -298.946,Y 259.403,Z -30.000,A 0.015,B 0.000,C 180.000},{X -303.931,Y 273.896,Z -30.000,A 0.015,B 0.000,C -180.000} C_DIS
CIRC {X -305.809,Y 276.807,Z -30.000,A 0.015,B 0.000,C -180.000},{X -309.083,Y 277.937,Z -30.000,A 0.015,B 0.000,C 180.000} C_DIS
LIN {X -338.669,Y 277.937,Z -30.000,A 0.015,B 0.000,C 180.000} C_DIS
CIRC {X -341.393,Y 276.808,Z -30.000,A 0.015,B 0.000,C -180.000},{X -342.521,Y 274.083,Z -30.000,A 0.015,B -0.000,C -180.000} C_DIS
LIN {X -342.517,Y 123.042,Z -30.000,A 0.015,B 0.000,C -180.000} C_DIS
CIRC {X -341.428,Y 119.511,Z -30.000,A 0.015,B -0.000,C -180.000},{X -338.540,Y 117.206,Z -30.000,A 0.015,B 0.000,C 180.000} C_DIS
CIRC {X -329.788,Y 113.404,Z -30.000,A 0.015,B 0.000,C 180.000},{X -321.327,Y 108.994,Z -30.000,A 0.015,B 0.000,C -180.000} C_DIS
CIRC {X -313.309,Y 103.801,Z -30.000,A 0.015,B 0.000,C 180.000},{X -305.957,Y 97.702,Z -30.000,A 0.015,B 0.000,C -180.000} C_DIS
CIRC {X -295.256,Y 85.948,Z -30.000,A 0.015,B 0.000,C 180.000},{X -286.589,Y 72.623,Z -30.000,A 0.015,B 0.000,C -180.000} C_DIS
LIN {X -271.141,Y 44.957,Z -30.000,A 0.015,B 0.000,C -180.000} C_DIS
CIRC {X -269.758,Y 42.311,Z -30.000,A 0.015,B -0.000,C -180.000},{X -268.598,Y 39.560,Z -30.000,A 0.015,B 0.000,C 180.000} C_DIS
CIRC {X -267.526,Y 36.776,Z -30.000,A 0.015,B 0.000,C -180.000},{X -266.401,Y 34.013,Z -30.000,A 0.015,B 0.000,C -180.000} C_DIS
CIRC {X -263.993,Y 31.093,Z -30.000,A 0.015,B -0.000,C -180.000},{X -260.370,Y 29.998,Z -30.000,A 0.015,B 0.000,C 180.000} C_DIS
LIN {X -133.129,Y 29.998,Z -30.000,A 0.015,B 0.000,C -180.000} C_DIS
CIRC {X -129.524,Y 31.085,Z -30.000,A 0.015,B 0.000,C 180.000},{X -127.122,Y 33.984,Z -30.000,A 0.015,B 0.000,C 180.000} C_DIS
CIRC {X -125.943,Y 36.864,Z -30.000,A 0.015,B 0.000,C 180.000},{X -124.824,Y 39.769,Z -30.000,A 0.015,B 0.000,C -180.000} C_DIS
CIRC {X -123.615,Y 42.639,Z -30.000,A 0.015,B 0.000,C 180.000},{X -122.170,Y 45.398,Z -30.000,A 0.015,B 0.000,C -180.000} C_DIS
LIN {X -103.145,Y 78.318,Z -30.000,A 0.015,B 0.000,C 180.000} C_DIS
CIRC {X -91.633,Y 93.868,Z -30.000,A 0.015,B 0.000,C -180.000},{X -76.921,Y 106.434,Z -30.000,A 0.015,B 0.000,C 180.000} C_DIS
CIRC {X -71.704,Y 109.638,Z -30.000,A 0.015,B 0.000,C 180.000},{X -66.233,Y 112.384,Z -30.000,A 0.015,B 0.000,C 180.000} C_DIS
CIRC {X -60.627,Y 114.832,Z -30.000,A 0.015,B -0.000,C 180.000},{X -54.972,Y 117.163,Z -30.000,A 0.015,B 0.000,C 180.000} C_DIS
CIRC {X -52.081,Y 119.492,Z -30.000,A 0.015,B 0.000,C 180.000},{X -50.993,Y 123.041,Z -30.000,A 0.015,B 0.000,C 180.000} C_DIS
LIN {X -50.997,Y 274.091,Z -30.000,A 0.015,B 0.000,C 180.000} C_DIS
CIRC {X -52.126,Y 276.815,Z -30.000,A 0.015,B -0.000,C 180.000},{X -54.850,Y 277.943,Z -30.000,A 0.015,B 0.000,C 180.000} C_DIS
LIN {X -84.477,Y 277.943,Z -30.000,A 0.015,B 0.000,C -180.000} C_DIS
CIRC {X -87.737,Y 276.809,Z -30.000,A 0.015,B 0.000,C -180.000},{X -89.591,Y 273.899,Z -30.000,A 0.015,B 0.000,C 180.000} C_DIS
CIRC {X -96.457,Y 255.094,Z -30.000,A 0.015,B 0.000,C 180.000},{X -107.514,Y 238.406,Z -30.000,A 0.015,B -0.000,C -180.000} C_DIS
CIRC {X -122.037,Y 224.653,Z -30.000,A 0.015,B 0.000,C -180.000},{X -139.211,Y 214.400,Z -30.000,A 0.015,B -0.000,C 180.000} C_DIS
CIRC {X -148.661,Y 210.647,Z -30.000,A 0.015,B 0.000,C 180.000},{X -158.439,Y 207.861,Z -30.000,A 0.015,B -0.000,C 180.000} C_DIS
CIRC {X -168.462,Y 206.135,Z -30.000,A 0.015,B 0.000,C -180.000},{X -178.617,Y 205.558,Z -30.000,A 0.015,B -0.000,C -180.000} C_DIS
LIN {X -217.274,Y 205.665,Z -30.000,A 0.015,B -0.000,C -180.000} C_DIS
CIRC {X -236.591,Y 208.002,Z -30.000,A 0.015,B -0.000,C 180.000},{X -254.868,Y 214.673,Z -30.000,A 0.015,B 0.000,C 180.000} C_DIS
CIRC {X -271.591,Y 225.242,Z -30.000,A 0.015,B 0.000,C 180.000},{X -285.909,Y 238.892,Z -30.000,A 0.015,B 0.000,C -180.000} C_DIS
CIRC {X -288.764,Y 242.396,Z -30.000,A 0.015,B -0.000,C 180.000},{X -291.428,Y 246.048,Z -30.000,A 0.015,B 0.000,C -180.000} C_DIS
CIRC {X -292.727,Y 250.220,Z -30.000,A 0.015,B 0.000,C -180.000},{X -291.431,Y 254.393,Z -30.000,A 0.015,B 0.000,C 180.000} C_DIS
CIRC {X -289.965,Y 258.449,Z -30.000,A 0.015,B 0.000,C 180.000},{X -290.671,Y 262.704,Z -30.000,A 0.015,B -0.000,C 180.000} C_DIS
CIRC {X -292.974,Y 268.553,Z -30.000,A 0.015,B -0.000,C 180.000},{X -294.744,Y 274.584,Z -30.000,A 0.015,B -0.000,C 180.000} C_DIS
CIRC {X -295.234,Y 276.745,Z -30.000,A 0.015,B -0.000,C -180.000},{X -295.645,Y 278.923,Z -30.000,A 0.015,B -0.000,C 180.000} C_DIS
CIRC {X -296.044,Y 281.102,Z -30.000,A 0.015,B -0.000,C 180.000},{X -296.500,Y 283.271,Z -30.000,A 0.015,B -0.000,C -180.000} C_DIS
CIRC {X -298.307,Y 286.169,Z -30.000,A 0.015,B 0.000,C -180.000},{X -301.530,Y 287.300,Z -30.000,A 0.015,B 0.000,C 180.000} C_DIS
LIN {X -348.031,Y 287.299,Z -30.000,A 0.015,B -0.000,C -180.000} C_DIS
CIRC {X -350.756,Y 286.170,Z -30.000,A 0.015,B 0.000,C 180.000},{X -351.884,Y 283.446,Z -30.000,A 0.015,B -0.000,C 180.000} C_DIS
LIN {X -351.880,Y 115.543,Z -30.000,A 0.015,B 0.000,C -180.000} C_DIS
CIRC {X -350.791,Y 112.341,Z -30.000,A 0.015,B 0.000,C 180.000},{X -347.977,Y 110.466,Z -30.000,A 0.015,B -0.000,C 180.000} C_DIS
CIRC {X -334.232,Y 105.410,Z -30.000,A 0.015,B 0.000,C 180.000},{X -321.654,Y 97.909,Z -30.000,A 0.015,B 0.000,C 180.000} C_DIS
CIRC {X -310.515,Y 88.435,Z -30.000,A 0.015,B 0.000,C 180.000},{X -300.908,Y 77.410,Z -30.000,A 0.015,B 0.000,C 180.000} C_DIS
LIN {X -279.119,Y 40.359,Z -30.000,A 0.015,B 0.000,C -180.000} C_DIS
CIRC {X -277.193,Y 36.597,Z -30.000,A 0.015,B 0.000,C 180.000},{X -275.650,Y 32.663,Z -30.000,A 0.015,B 0.000,C -180.000} C_DIS
CIRC {X -274.293,Y 28.666,Z -30.000,A 0.015,B 0.000,C 180.000},{X -272.912,Y 24.677,Z -30.000,A 0.015,B 0.000,C -180.000} C_DIS
CIRC {X -270.710,Y 21.748,Z -30.000,A 0.015,B 0.000,C -180.000},{X -267.219,Y 20.635,Z -30.000,A 0.015,B 0.000,C 180.000} C_DIS
LIN {X -126.295,Y 20.635,Z -30.000,A 0.015,B 0.000,C -180.000} C_DIS
CIRC {X -122.805,Y 21.746,Z -30.000,A 0.015,B 0.000,C 180.000},{X -120.600,Y 24.670,Z -30.000,A 0.015,B 0.000,C 180.000} C_DIS
CIRC {X -119.173,Y 28.770,Z -30.000,A 0.015,B -0.000,C -180.000},{X -117.772,Y 32.879,Z -30.000,A 0.015,B 0.000,C -180.000} C_DIS
CIRC {X -116.181,Y 36.923,Z -30.000,A 0.015,B 0.000,C -180.000},{X -114.195,Y 40.790,Z -30.000,A 0.015,B 0.000,C -180.000} C_DIS
LIN {X -96.233,Y 72.150,Z -30.000,A 0.015,B 0.000,C -180.000} C_DIS
CIRC {X -85.493,Y 86.832,Z -30.000,A 0.015,B -0.000,C 180.000},{X -71.684,Y 98.673,Z -30.000,A 0.015,B 0.000,C -180.000} C_DIS
CIRC {X -65.542,Y 102.435,Z -30.000,A 0.015,B 0.000,C -180.000},{X -59.093,Y 105.642,Z -30.000,A 0.015,B 0.000,C 180.000} C_DIS
CIRC {X -52.405,Y 108.311,Z -30.000,A 0.015,B 0.000,C -180.000},{X -45.536,Y 110.469,Z -30.000,A 0.015,B 0.000,C 180.000} C_DIS
CIRC {X -42.718,Y 112.367,Z -30.000,A 0.015,B 0.000,C -180.000},{X -41.630,Y 115.586,Z -30.000,A 0.015,B -0.000,C -180.000} C_DIS
LIN {X -41.635,Y 283.453,Z -30.000,A 0.015,B 0.000,C 180.000} C_DIS
CIRC {X -42.763,Y 286.178,Z -30.000,A 0.015,B 0.000,C -180.000},{X -45.488,Y 287.306,Z -30.000,A 0.015,B 0.000,C -180.000} C_DIS
LIN {X -91.924,Y 287.305,Z -30.000,A 0.015,B 0.000,C -180.000} C_DIS
CIRC {X -95.150,Y 286.184,Z -30.000,A 0.015,B -0.000,C -180.000},{X -96.984,Y 283.304,Z -30.000,A 0.015,B 0.000,C 180.000} C_DIS
LIN {X -99.671,Y 271.790,Z -30.000,A 0.015,B 0.000,C -180.000} C_DIS
CIRC {X -101.400,Y 266.122,Z -30.000,A 0.015,B 0.000,C -180.000},{X -103.903,Y 260.751,Z -30.000,A 0.015,B 0.000,C 180.000} C_DIS
CIRC {X -115.593,Y 244.218,Z -30.000,A 0.015,B 0.000,C -180.000},{X -130.587,Y 230.611,Z -30.000,A 0.015,B 0.000,C -180.000} C_DIS
CIRC {X -148.370,Y 220.847,Z -30.000,A 0.015,B 0.000,C 180.000},{X -168.022,Y 215.813,Z -30.000,A 0.015,B 0.000,C 180.000} C_DIS
CIRC {X -170.663,Y 215.494,Z -30.000,A 0.015,B 0.000,C -180.000},{X -173.306,Y 215.201,Z -30.000,A 0.015,B -0.000,C -180.000} C_DIS
CIRC {X -175.957,Y 214.990,Z -30.000,A 0.015,B 0.000,C 180.000},{X -178.617,Y 214.920,Z -30.000,A 0.015,B -0.000,C 180.000} C_DIS
LIN {X -215.118,Y 214.777,Z -30.000,A 0.015,B 0.000,C 180.000} C_DIS
CIRC {X -233.386,Y 216.799,Z -30.000,A 0.015,B 0.000,C 180.000},{X -250.672,Y 223.042,Z -30.000,A 0.015,B 0.000,C 180.000} C_DIS
CIRC {X -265.479,Y 232.240,Z -30.000,A 0.015,B 0.000,C 180.000},{X -278.373,Y 243.969,Z -30.000,A 0.015,B 0.000,C 180.000} C_DIS
CIRC {X -285.276,Y 252.842,Z -30.000,A 0.015,B 0.000,C 180.000},{X -290.671,Y 262.704,Z -30.000,A 0.015,B 0.000,C 180.000} C_DIS
CIRC {X -291.206,Y 267.329,Z -30.000,A 0.015,B 0.000,C 180.000},{X -288.998,Y 271.428,Z -30.000,A 0.015,B 0.000,C 180.000} C_DIS
CIRC {X -286.633,Y 275.366,Z -30.000,A 0.015,B 0.000,C 180.000},{X -286.522,Y 279.958,Z -30.000,A 0.015,B 0.000,C 180.000} C_DIS
CIRC {X -287.846,Y 286.378,Z -30.000,A 0.015,B 0.000,C 180.000},{X -288.775,Y 292.867,Z -30.000,A 0.015,B 0.000,C 180.000} C_DIS
CIRC {X -290.173,Y 295.575,Z -30.000,A 0.015,B 0.000,C 180.000},{X -293.021,Y 296.663,Z -30.000,A 0.015,B 0.000,C 180.000} C_DIS
LIN {X -357.394,Y 296.661,Z -30.000,A 0.015,B 0.000,C 180.000} C_DIS
CIRC {X -360.119,Y 295.533,Z -30.000,A 0.015,B 0.000,C 180.000},{X -361.247,Y 292.808,Z -30.000,A 0.015,B 0.000,C 180.000} C_DIS
LIN {X -361.242,Y 107.508,Z -30.000,A 0.015,B -0.000,C -180.000} C_DIS
CIRC {X -360.158,Y 104.506,Z -30.000,A 0.015,B 0.000,C -180.000},{X -357.405,Y 102.890,Z -30.000,A 0.015,B -0.000,C -180.000} C_DIS
CIRC {X -352.804,Y 101.948,Z -30.000,A 0.015,B 0.000,C 180.000},{X -348.239,Y 100.846,Z -30.000,A 0.015,B 0.000,C -180.000} C_DIS
CIRC {X -343.741,Y 99.488,Z -30.000,A 0.015,B 0.000,C -180.000},{X -339.360,Y 97.787,Z -30.000,A 0.015,B 0.000,C -180.000} C_DIS
CIRC {X -321.769,Y 86.742,Z -30.000,A 0.015,B 0.000,C 180.000},{X -308.285,Y 70.942,Z -30.000,A 0.015,B 0.000,C -180.000} C_DIS
LIN {X -287.216,Y 35.694,Z -30.000,A 0.015,B 0.000,C 180.000} C_DIS
CIRC {X -284.731,Y 30.822,Z -30.000,A 0.015,B 0.000,C -180.000},{X -282.753,Y 25.724,Z -30.000,A 0.015,B 0.000,C 180.000} C_DIS
CIRC {X -281.170,Y 20.495,Z -30.000,A 0.015,B 0.000,C -180.000},{X -279.852,Y 15.193,Z -30.000,A 0.015,B 0.000,C 180.000} C_DIS
CIRC {X -278.098,Y 12.374,Z -30.000,A 0.015,B -0.000,C -180.000},{X -274.966,Y 11.273,Z -30.000,A 0.015,B 0.000,C -180.000} C_DIS
LIN {X -118.610,Y 11.273,Z -30.000,A 0.015,B 0.000,C 180.000} C_DIS
CIRC {X -115.430,Y 12.390,Z -30.000,A 0.015,B 0.000,C -180.000},{X -113.647,Y 15.250,Z -30.000,A 0.015,B 0.000,C 180.000} C_DIS
CIRC {X -109.313,Y 29.242,Z -30.000,A 0.015,B 0.000,C 180.000},{X -102.788,Y 42.357,Z -30.000,A 0.015,B 0.000,C -180.000} C_DIS
LIN {X -87.945,Y 67.506,Z -30.000,A 0.015,B 0.000,C -180.000} C_DIS
CIRC {X -80.436,Y 78.016,Z -30.000,A 0.015,B -0.000,C 180.000},{X -71.054,Y 86.894,Z -30.000,A 0.015,B 0.000,C 180.000} C_DIS
CIRC {X -60.384,Y 94.119,Z -30.000,A 0.015,B 0.000,C -180.000},{X -48.854,Y 99.871,Z -30.000,A 0.015,B -0.000,C -180.000} C_DIS
CIRC {X -45.655,Y 101.005,Z -30.000,A 0.015,B 0.000,C 180.000},{X -42.348,Y 101.772,Z -30.000,A 0.015,B 0.000,C 180.000} C_DIS
LIN {X -36.210,Y 102.838,Z -30.000,A 0.015,B 0.000,C 180.000} C_DIS
CIRC {X -33.384,Y 104.463,Z -30.000,A 0.015,B 0.000,C 180.000},{X -32.267,Y 107.525,Z -30.000,A 0.015,B 0.000,C 180.000} C_DIS
LIN {X -32.272,Y 292.816,Z -30.000,A 0.015,B 0.000,C 180.000} C_DIS
CIRC {X -33.401,Y 295.541,Z -30.000,A 0.015,B 0.000,C -180.000},{X -36.125,Y 296.669,Z -30.000,A 0.015,B -0.000,C 180.000} C_DIS
LIN {X -100.526,Y 296.668,Z -30.000,A 0.015,B 0.000,C 180.000} C_DIS
CIRC {X -103.358,Y 295.579,Z -30.000,A 0.015,B 0.000,C 180.000},{X -104.732,Y 292.875,Z -30.000,A 0.015,B 0.000,C 180.000} C_DIS
CIRC {X -106.482,Y 282.436,Z -30.000,A 0.015,B 0.000,C -180.000},{X -109.525,Y 272.297,Z -30.000,A 0.015,B -0.000,C -180.000} C_DIS
CIRC {X -113.874,Y 262.642,Z -30.000,A 0.015,B 0.000,C 180.000},{X -119.508,Y 253.675,Z -30.000,A 0.015,B 0.000,C 180.000} C_DIS
CIRC {X -128.957,Y 243.240,Z -30.000,A 0.015,B -0.000,C 180.000},{X -140.392,Y 235.028,Z -30.000,A 0.015,B 0.000,C 180.000} C_DIS
CIRC {X -153.148,Y 229.142,Z -30.000,A 0.015,B -0.000,C 180.000},{X -166.711,Y 225.482,Z -30.000,A 0.015,B -0.000,C 180.000} C_DIS
CIRC {X -178.698,Y 223.984,Z -30.000,A 0.015,B 0.000,C -180.000},{X -190.776,Y 223.803,Z -30.000,A 0.015,B -0.000,C -180.000} C_DIS
CIRC {X -202.834,Y 224.163,Z -30.000,A 0.015,B 0.000,C 180.000},{X -214.895,Y 224.283,Z -30.000,A 0.015,B 0.000,C 180.000} C_DIS
CIRC {X -233.068,Y 226.619,Z -30.000,A 0.015,B 0.000,C 180.000},{X -250.057,Y 233.477,Z -30.000,A 0.015,B 0.000,C 180.000} C_DIS
CIRC {X -264.906,Y 244.151,Z -30.000,A 0.015,B 0.000,C -180.000},{X -277.019,Y 257.849,Z -30.000,A 0.015,B 0.000,C 180.000} C_DIS
CIRC {X -281.746,Y 265.903,Z -30.000,A 0.015,B 0.000,C 180.000},{X -285.101,Y 274.618,Z -30.000,A 0.015,B 0.000,C 180.000} C_DIS
CIRC {X -285.846,Y 277.279,Z -30.000,A 0.015,B 0.000,C 180.000},{X -286.522,Y 279.958,Z -30.000,A 0.015,B 0.000,C -180.000} C_DIS
CIRC {X -286.222,Y 284.311,Z -30.000,A 0.015,B 0.000,C 180.000},{X -283.498,Y 287.719,Z -30.000,A 0.015,B 0.000,C 180.000} C_DIS
CIRC {X -280.644,Y 290.934,Z -30.000,A 0.015,B 0.000,C -180.000},{X -279.687,Y 295.125,Z -30.000,A 0.015,B -0.000,C -180.000} C_DIS
CIRC {X -279.677,Y 298.761,Z -30.000,A 0.015,B 0.000,C -180.000},{X -279.453,Y 302.390,Z -30.000,A 0.015,B 0.000,C -180.000} C_DIS
CIRC {X -280.310,Y 304.940,Z -30.000,A 0.015,B 0.000,C 180.000},{X -282.772,Y 306.026,Z -30.000,A 0.015,B 0.000,C 180.000} C_DIS
LIN {X -366.757,Y 306.024,Z -30.000,A 0.015,B 0.000,C -180.000} C_DIS
CIRC {X -369.482,Y 304.895,Z -30.000,A 0.015,B 0.000,C 180.000},{X -370.610,Y 302.171,Z -30.000,A 0.015,B -0.000,C 180.000} C_DIS
LIN {X -370.604,Y 98.583,Z -30.000,A 0.015,B 0.000,C -180.000} C_DIS
CIRC {X -369.524,Y 95.840,Z -30.000,A 0.015,B -0.000,C 180.000},{X -366.864,Y 94.569,Z -30.000,A 0.015,B 0.000,C 180.000} C_DIS
CIRC {X -360.777,Y 93.933,Z -30.000,A 0.015,B 0.000,C 180.000},{X -354.746,Y 92.891,Z -30.000,A 0.015,B 0.000,C 180.000} C_DIS
CIRC {X -348.820,Y 91.342,Z -30.000,A 0.015,B 0.000,C -180.000},{X -343.083,Y 89.197,Z -30.000,A 0.015,B 0.000,C -180.000} C_DIS
CIRC {X -326.797,Y 78.843,Z -30.000,A 0.015,B 0.000,C -180.000},{X -314.518,Y 63.956,Z -30.000,A 0.015,B -0.000,C -180.000} C_DIS
LIN {X -295.328,Y 31.019,Z -30.000,A 0.015,B 0.000,C -180.000} C_DIS
CIRC {X -292.370,Y 25.068,Z -30.000,A 0.015,B 0.000,C 180.000},{X -290.162,Y 18.800,Z -30.000,A 0.015,B 0.000,C 180.000} C_DIS
CIRC {X -288.639,Y 12.337,Z -30.000,A 0.015,B -0.000,C 180.000},{X -287.715,Y 5.762,Z -30.000,A 0.015,B 0.000,C 180.000} C_DIS
CIRC {X -286.344,Y 3.017,Z -30.000,A 0.015,B 0.000,C 180.000},{X -283.484,Y 1.910,Z -30.000,A 0.015,B 0.000,C -180.000} C_DIS
LIN {X -110.057,Y 1.910,Z -30.000,A 0.015,B 0.000,C -180.000} C_DIS
CIRC {X -107.145,Y 3.038,Z -30.000,A 0.015,B 0.000,C -180.000},{X -105.753,Y 5.832,Z -30.000,A 0.015,B 0.000,C 180.000} C_DIS
CIRC {X -104.814,Y 12.498,Z -30.000,A 0.015,B -0.000,C 180.000},{X -103.253,Y 19.047,Z -30.000,A 0.015,B -0.000,C 180.000} C_DIS
CIRC {X -100.996,Y 25.395,Z -30.000,A 0.015,B 0.000,C -180.000},{X -97.985,Y 31.422,Z -30.000,A 0.015,B 0.000,C -180.000} C_DIS
CIRC {X -91.937,Y 42.134,Z -30.000,A 0.015,B 0.000,C 180.000},{X -86.105,Y 52.966,Z -30.000,A 0.015,B 0.000,C -180.000} C_DIS
CIRC {X -79.720,Y 63.507,Z -30.000,A 0.015,B -0.000,C 180.000},{X -72.102,Y 73.195,Z -30.000,A 0.015,B 0.000,C -180.000} C_DIS
CIRC {X -63.243,Y 81.444,Z -30.000,A 0.015,B -0.000,C -180.000},{X -53.001,Y 87.893,Z -30.000,A 0.015,B 0.000,C 180.000} C_DIS
CIRC {X -41.714,Y 92.275,Z -30.000,A 0.015,B 0.000,C 180.000},{X -29.790,Y 94.381,Z -30.000,A 0.015,B 0.000,C -180.000} C_DIS
CIRC {X -29.019,Y 94.428,Z -30.000,A 0.015,B 0.000,C 180.000},{X -28.248,Y 94.451,Z -30.000,A 0.015,B -0.000,C 180.000} C_DIS
CIRC {X -27.476,Y 94.474,Z -30.000,A 0.015,B 0.000,C 180.000},{X -26.706,Y 94.522,Z -30.000,A 0.015,B 0.000,C 180.000} C_DIS
CIRC {X -24.001,Y 95.830,Z -30.000,A 0.015,B 0.000,C 180.000},{X -22.904,Y 98.628,Z -30.000,A 0.015,B 0.000,C 180.000} C_DIS
LIN {X -22.910,Y 302.179,Z -30.000,A 0.015,B -0.000,C 180.000} C_DIS
CIRC {X -24.039,Y 304.904,Z -30.000,A 0.015,B 0.000,C -180.000},{X -26.763,Y 306.032,Z -30.000,A 0.015,B 0.000,C 180.000} C_DIS
LIN {X -110.777,Y 306.030,Z -30.000,A 0.015,B 0.000,C 180.000} C_DIS
CIRC {X -113.223,Y 304.936,Z -30.000,A 0.015,B 0.000,C 180.000},{X -114.039,Y 302.384,Z -30.000,A 0.015,B 0.000,C 180.000} C_DIS
CIRC {X -115.309,Y 282.538,Z -30.000,A 0.015,B -0.000,C -180.000},{X -123.297,Y 264.326,Z -30.000,A 0.015,B 0.000,C -180.000} C_DIS
CIRC {X -136.434,Y 249.547,Z -30.000,A 0.015,B 0.000,C 180.000},{X -153.115,Y 238.929,Z -30.000,A 0.015,B 0.000,C 180.000} C_DIS
CIRC {X -158.142,Y 236.983,Z -30.000,A 0.015,B 0.000,C -180.000},{X -163.362,Y 235.640,Z -30.000,A 0.015,B 0.000,C 180.000} C_DIS
CIRC {X -168.660,Y 234.697,Z -30.000,A 0.015,B 0.000,C -180.000},{X -173.987,Y 233.935,Z -30.000,A 0.015,B 0.000,C 180.000} C_DIS
LIN {X -214.895,Y 233.645,Z -30.000,A 0.015,B 0.000,C 180.000} C_DIS
CIRC {X -240.664,Y 238.887,Z -30.000,A 0.015,B 0.000,C 180.000},{X -262.337,Y 253.778,Z -30.000,A 0.015,B 0.000,C -180.000} C_DIS
CIRC {X -274.890,Y 272.824,Z -30.000,A 0.015,B 0.000,C 180.000},{X -279.687,Y 295.125,Z -30.000,A 0.015,B 0.000,C 180.000} C_DIS
CIRC {X -278.457,Y 299.319,Z -30.000,A 0.015,B 0.000,C 180.000},{X -275.009,Y 302.006,Z -30.000,A 0.015,B -0.000,C 180.000} C_DIS
CIRC {X -271.473,Y 304.450,Z -30.000,A 0.015,B 0.000,C -180.000},{X -269.573,Y 308.306,Z -30.000,A 0.015,B 0.000,C 180.000} C_DIS
CIRC {X -269.279,Y 309.832,Z -30.000,A 0.015,B 0.000,C 180.000},{X -269.024,Y 311.366,Z -30.000,A 0.015,B -0.000,C 180.000} C_DIS
CIRC {X -269.759,Y 313.930,Z -30.000,A 0.015,B -0.000,C 180.000},{X -272.182,Y 315.044,Z -30.000,A 0.015,B -0.000,C -180.000} C_DIS
LIN {X -375.775,Y 315.041,Z -30.000,A 0.015,B 0.000,C -180.000} C_DIS
CIRC {X -378.500,Y 313.913,Z -30.000,A 0.015,B 0.000,C 180.000},{X -379.628,Y 311.188,Z -30.000,A 0.015,B -0.000,C -180.000} C_DIS
LIN {X -379.622,Y 88.724,Z -30.000,A 0.015,B -0.000,C 180.000} C_DIS
CIRC {X -378.548,Y 86.294,Z -30.000,A 0.015,B 0.000,C 180.000},{X -376.027,Y 85.453,Z -30.000,A 0.015,B 0.000,C -180.000} C_DIS
CIRC {X -355.278,Y 83.749,Z -30.000,A 0.015,B -0.000,C 180.000},{X -336.393,Y 74.988,Z -30.000,A 0.015,B 0.000,C -180.000} C_DIS
CIRC {X -332.585,Y 71.932,Z -30.000,A 0.015,B 0.000,C -180.000},{X -329.197,Y 68.416,Z -30.000,A 0.015,B 0.000,C -180.000} C_DIS
CIRC {X -326.103,Y 64.652,Z -30.000,A 0.015,B 0.000,C 180.000},{X -323.125,Y 60.794,Z -30.000,A 0.015,B 0.000,C 180.000} C_DIS
LIN {X -303.142,Y 26.516,Z -30.000,A 0.015,B 0.000,C -180.000} C_DIS
CIRC {X -300.351,Y 20.805,Z -30.000,A 0.015,B 0.000,C -180.000},{X -298.363,Y 14.767,Z -30.000,A 0.015,B 0.000,C 180.000} C_DIS
CIRC {X -297.064,Y 8.553,Z -30.000,A 0.015,B 0.000,C 180.000},{X -296.310,Y 2.250,Z -30.000,A 0.015,B 0.000,C 180.000} C_DIS
CIRC {X -296.264,Y 0.833,Z -30.000,A 0.015,B -0.000,C 180.000},{X -296.340,Y -0.584,Z -30.000,A 0.015,B -0.000,C -180.000} C_DIS
CIRC {X -296.460,Y -1.996,Z -30.000,A 0.015,B 0.000,C 180.000},{X -296.543,Y -3.410,Z -30.000,A 0.015,B -0.000,C 180.000} C_DIS
CIRC {X -295.569,Y -6.014,Z -30.000,A 0.015,B 0.000,C 180.000},{X -293.013,Y -7.108,Z -30.000,A 0.015,B -0.000,C -180.000} C_DIS
LIN {X -100.499,Y -7.108,Z -30.000,A 0.015,B 0.000,C -180.000} C_DIS
CIRC {X -97.943,Y -6.014,Z -30.000,A 0.015,B 0.000,C 180.000},{X -96.969,Y -3.410,Z -30.000,A 0.015,B 0.000,C 180.000} C_DIS
CIRC {X -97.084,Y 1.120,Z -30.000,A 0.015,B 0.000,C 180.000},{X -97.012,Y 5.652,Z -30.000,A 0.015,B 0.000,C -180.000} C_DIS
CIRC {X -96.504,Y 10.167,Z -30.000,A 0.015,B 0.000,C 180.000},{X -95.324,Y 14.555,Z -30.000,A 0.015,B -0.000,C -180.000} C_DIS
CIRC {X -94.197,Y 17.709,Z -30.000,A 0.015,B -0.000,C 180.000},{X -93.038,Y 20.852,Z -30.000,A 0.015,B 0.000,C 180.000} C_DIS
CIRC {X -91.733,Y 23.940,Z -30.000,A 0.015,B 0.000,C 180.000},{X -90.177,Y 26.909,Z -30.000,A 0.015,B 0.000,C 180.000} C_DIS
LIN {X -69.868,Y 61.520,Z -30.000,A 0.015,B 0.000,C 180.000} C_DIS
CIRC {X -62.893,Y 69.398,Z -30.000,A 0.015,B 0.000,C 180.000},{X -54.987,Y 76.342,Z -30.000,A 0.015,B 0.000,C -180.000} C_DIS
CIRC {X -45.894,Y 81.750,Z -30.000,A 0.015,B 0.000,C 180.000},{X -35.767,Y 84.811,Z -30.000,A 0.015,B -0.000,C -180.000} C_DIS
CIRC {X -31.222,Y 85.436,Z -30.000,A 0.015,B 0.000,C 180.000},{X -26.645,Y 85.741,Z -30.000,A 0.015,B 0.000,C 180.000} C_DIS
CIRC {X -22.059,Y 85.741,Z -30.000,A 0.015,B 0.000,C 180.000},{X -17.481,Y 85.453,Z -30.000,A 0.015,B 0.000,C 180.000} C_DIS
CIRC {X -14.961,Y 86.293,Z -30.000,A 0.015,B 0.000,C -180.000},{X -13.886,Y 88.723,Z -30.000,A 0.015,B 0.000,C -180.000} C_DIS
LIN {X -13.892,Y 311.197,Z -30.000,A 0.015,B -0.000,C 180.000} C_DIS
CIRC {X -15.021,Y 313.922,Z -30.000,A 0.015,B 0.000,C -180.000},{X -17.745,Y 315.050,Z -30.000,A 0.015,B 0.000,C 180.000} C_DIS
LIN {X -121.329,Y 315.048,Z -30.000,A 0.015,B 0.000,C -180.000} C_DIS
CIRC {X -123.733,Y 313.946,Z -30.000,A 0.015,B 0.000,C -180.000},{X -124.470,Y 311.406,Z -30.000,A 0.015,B 0.000,C 180.000} C_DIS
CIRC {X -123.681,Y 306.366,Z -30.000,A 0.015,B 0.000,C -180.000},{X -122.810,Y 301.340,Z -30.000,A 0.015,B 0.000,C 180.000} C_DIS
CIRC {X -122.418,Y 296.226,Z -30.000,A 0.015,B 0.000,C -180.000},{X -123.081,Y 291.141,Z -30.000,A 0.015,B 0.000,C 180.000} C_DIS
CIRC {X -125.142,Y 283.593,Z -30.000,A 0.015,B -0.000,C 180.000},{X -127.709,Y 276.202,Z -30.000,A 0.015,B 0.000,C 180.000} C_DIS
CIRC {X -131.146,Y 269.147,Z -30.000,A 0.015,B 0.000,C -180.000},{X -135.727,Y 262.774,Z -30.000,A 0.015,B -0.000,C 180.000} C_DIS
CIRC {X -143.171,Y 255.523,Z -30.000,A 0.015,B 0.000,C -180.000},{X -151.794,Y 249.723,Z -30.000,A 0.015,B 0.000,C -180.000} C_DIS
CIRC {X -161.338,Y 245.601,Z -30.000,A 0.015,B 0.000,C -180.000},{X -171.484,Y 243.339,Z -30.000,A 0.015,B 0.000,C -180.000} C_DIS
LIN {X -214.895,Y 242.663,Z -30.000,A 0.015,B 0.000,C 180.000} C_DIS
CIRC {X -228.706,Y 244.475,Z -30.000,A 0.015,B 0.000,C -180.000},{X -241.582,Y 249.787,Z -30.000,A 0.015,B -0.000,C -180.000} C_DIS
CIRC {X -252.801,Y 257.983,Z -30.000,A 0.015,B 0.000,C 180.000},{X -261.978,Y 268.414,Z -30.000,A 0.015,B 0.000,C -180.000} C_DIS
CIRC {X -269.322,Y 284.154,Z -30.000,A 0.015,B 0.000,C 180.000},{X -270.796,Y 301.461,Z -30.000,A 0.015,B 0.000,C 180.000} C_DIS
CIRC {X -270.487,Y 303.959,Z -30.000,A 0.015,B 0.000,C 180.000},{X -269.992,Y 306.428,Z -30.000,A 0.015,B -0.000,C 180.000} C_DIS
CIRC {X -269.775,Y 307.365,Z -30.000,A 0.015,B -0.000,C 180.000},{X -269.573,Y 308.306,Z -30.000,A 0.015,B 0.000,C 180.000} C_DIS
CIRC {X -267.636,Y 311.812,Z -30.000,A 0.015,B 0.000,C -180.000},{X -264.053,Y 313.602,Z -30.000,A 0.015,B 0.000,C -180.000} C_DIS
CIRC {X -260.429,Y 315.148,Z -30.000,A 0.015,B 0.000,C -180.000},{X -257.939,Y 318.201,Z -30.000,A 0.015,B -0.000,C -180.000} C_DIS
CIRC {X -257.407,Y 319.288,Z -30.000,A 0.015,B 0.000,C -180.000},{X -256.845,Y 320.361,Z -30.000,A 0.015,B 0.000,C 180.000} C_DIS
CIRC {X -256.894,Y 322.622,Z -30.000,A 0.015,B -0.000,C 180.000},{X -258.860,Y 323.738,Z -30.000,A 0.015,B 0.000,C 180.000} C_DIS
LIN {X -384.470,Y 323.735,Z -30.000,A 0.015,B -0.000,C 180.000} C_DIS
CIRC {X -387.194,Y 322.607,Z -30.000,A 0.015,B 0.000,C -180.000},{X -388.322,Y 319.882,Z -30.000,A 0.015,B -0.000,C -180.000} C_DIS
LIN {X -388.316,Y 77.008,Z -30.000,A 0.015,B -0.000,C -180.000} C_DIS
CIRC {X -387.194,Y 74.772,Z -30.000,A 0.015,B 0.000,C -180.000},{X -384.731,Y 74.335,Z -30.000,A 0.015,B 0.000,C -180.000} C_DIS
CIRC {X -382.019,Y 75.197,Z -30.000,A 0.015,B -0.000,C -180.000},{X -379.342,Y 76.158,Z -30.000,A 0.015,B 0.000,C 180.000} C_DIS
CIRC {X -376.595,Y 76.937,Z -30.000,A 0.015,B 0.000,C -180.000},{X -373.755,Y 77.231,Z -30.000,A 0.015,B -0.000,C 180.000} C_DIS
CIRC {X -364.532,Y 76.762,Z -30.000,A 0.015,B 0.000,C 180.000},{X -355.457,Y 75.055,Z -30.000,A 0.015,B -0.000,C -180.000} C_DIS
CIRC {X -346.827,Y 71.629,Z -30.000,A 0.015,B 0.000,C -180.000},{X -339.307,Y 66.182,Z -30.000,A 0.015,B 0.000,C 180.000} C_DIS
CIRC {X -336.380,Y 63.314,Z -30.000,A 0.015,B 0.000,C -180.000},{X -333.595,Y 60.308,Z -30.000,A 0.015,B -0.000,C -180.000} C_DIS
CIRC {X -331.038,Y 57.102,Z -30.000,A 0.015,B 0.000,C -180.000},{X -328.815,Y 53.655,Z -30.000,A 0.015,B 0.000,C -180.000} C_DIS
LIN {X -308.021,Y 16.233,Z -30.000,A 0.015,B 0.000,C -180.000} C_DIS
CIRC {X -305.835,Y 9.293,Z -30.000,A 0.015,B -0.000,C 180.000},{X -304.940,Y 2.073,Z -30.000,A 0.015,B 0.000,C -180.000} C_DIS
CIRC {X -305.168,Y -5.185,Z -30.000,A 0.015,B -0.000,C 180.000},{X -306.320,Y -12.353,Z -30.000,A 0.015,B 0.000,C 180.000} C_DIS
CIRC {X -305.773,Y -14.740,Z -30.000,A 0.015,B 0.000,C 180.000},{X -303.567,Y -15.802,Z -30.000,A 0.015,B 0.000,C -180.000} C_DIS
LIN {X -89.945,Y -15.802,Z -30.000,A 0.015,B -0.000,C 180.000} C_DIS
CIRC {X -87.739,Y -14.740,Z -30.000,A 0.015,B -0.000,C -180.000},{X -87.192,Y -12.353,Z -30.000,A 0.015,B 0.000,C 180.000} C_DIS
CIRC {X -88.165,Y -6.994,Z -30.000,A 0.015,B -0.000,C -180.000},{X -88.669,Y -1.570,Z -30.000,A 0.015,B 0.000,C -180.000} C_DIS
CIRC {X -88.583,Y 3.883,Z -30.000,A 0.015,B 0.000,C -180.000},{X -87.794,Y 9.280,Z -30.000,A 0.015,B 0.000,C 180.000} C_DIS
CIRC {X -86.998,Y 12.300,Z -30.000,A 0.015,B 0.000,C 180.000},{X -85.917,Y 15.230,Z -30.000,A 0.015,B 0.000,C -180.000} C_DIS
LIN {X -83.712,Y 20.429,Z -30.000,A 0.015,B 0.000,C -180.000} C_DIS
LIN {X -64.504,Y 53.959,Z -30.000,A 0.015,B -0.000,C 180.000} C_DIS
CIRC {X -57.167,Y 63.427,Z -30.000,A 0.015,B 0.000,C 180.000},{X -47.568,Y 70.592,Z -30.000,A 0.015,B -0.000,C -180.000} C_DIS
CIRC {X -36.567,Y 75.227,Z -30.000,A 0.015,B -0.000,C -180.000},{X -24.832,Y 77.413,Z -30.000,A 0.015,B 0.000,C -180.000} C_DIS
CIRC {X -20.710,Y 77.369,Z -30.000,A 0.015,B 0.000,C 180.000},{X -16.659,Y 76.606,Z -30.000,A 0.015,B 0.000,C -180.000} C_DIS
CIRC {X -12.710,Y 75.477,Z -30.000,A 0.015,B 0.000,C -180.000},{X -8.773,Y 74.310,Z -30.000,A 0.015,B 0.000,C 180.000} C_DIS
CIRC {X -6.314,Y 74.739,Z -30.000,A 0.015,B 0.000,C 180.000},{X -5.192,Y 76.970,Z -30.000,A 0.015,B -0.000,C 180.000} C_DIS
LIN {X -5.199,Y 319.891,Z -30.000,A 0.015,B 0.000,C -180.000} C_DIS
CIRC {X -6.327,Y 322.616,Z -30.000,A 0.015,B -0.000,C -180.000},{X -9.052,Y 323.744,Z -30.000,A 0.015,B 0.000,C 180.000} C_DIS
LIN {X -134.639,Y 323.741,Z -30.000,A 0.015,B -0.000,C 180.000} C_DIS
CIRC {X -136.609,Y 322.624,Z -30.000,A 0.015,B 0.000,C 180.000},{X -136.662,Y 320.361,Z -30.000,A 0.015,B 0.000,C 180.000} C_DIS
CIRC {X -134.147,Y 314.943,Z -30.000,A 0.015,B 0.000,C 180.000},{X -132.275,Y 309.271,Z -30.000,A 0.015,B 0.000,C -180.000} C_DIS
CIRC {X -131.182,Y 303.392,Z -30.000,A 0.015,B 0.000,C -180.000},{X -131.006,Y 297.414,Z -30.000,A 0.015,B -0.000,C 180.000} C_DIS
CIRC {X -133.649,Y 283.530,Z -30.000,A 0.015,B 0.000,C 180.000},{X -140.036,Y 270.923,Z -30.000,A 0.015,B 0.000,C 180.000} C_DIS
CIRC {X -149.914,Y 260.752,Z -30.000,A 0.015,B 0.000,C 180.000},{X -162.512,Y 254.246,Z -30.000,A 0.015,B 0.000,C 180.000} C_DIS
CIRC {X -166.450,Y 253.089,Z -30.000,A 0.015,B -0.000,C 180.000},{X -170.450,Y 252.166,Z -30.000,A 0.015,B 0.000,C 180.000} C_DIS
CIRC {X -174.513,Y 251.560,Z -30.000,A 0.015,B 0.000,C -180.000},{X -178.617,Y 251.357,Z -30.000,A 0.015,B -0.000,C -180.000} C_DIS
LIN {X -220.943,Y 251.965,Z -30.000,A 0.015,B -0.000,C 180.000} C_DIS
CIRC {X -241.941,Y 259.957,Z -30.000,A 0.015,B 0.000,C -180.000},{X -256.925,Y 276.698,Z -30.000,A 0.015,B 0.000,C 180.000} C_DIS
CIRC {X -262.368,Y 297.329,Z -30.000,A 0.015,B 0.000,C -180.000},{X -257.939,Y 318.201,Z -30.000,A 0.015,B -0.000,C 180.000} C_DIS
CIRC {X -255.525,Y 320.805,Z -30.000,A 0.015,B 0.000,C 180.000},{X -252.054,Y 321.558,Z -30.000,A 0.015,B 0.000,C 180.000} C_DIS
CIRC {X -248.601,Y 322.122,Z -30.000,A 0.015,B -0.000,C 180.000},{X -245.853,Y 324.289,Z -30.000,A 0.015,B 0.000,C -180.000} C_DIS
CIRC {X -244.170,Y 326.439,Z -30.000,A 0.015,B 0.000,C 180.000},{X -242.424,Y 328.539,Z -30.000,A 0.015,B 0.000,C 180.000} C_DIS
LIN {X -242.271,Y 328.704,Z -30.000,A 0.015,B 0.000,C 180.000} C_DIS
LIN {X -242.114,Y 328.865,Z -30.000,A 0.015,B 0.000,C 180.000} C_DIS
CIRC {X -241.785,Y 330.789,Z -30.000,A 0.015,B 0.000,C -180.000},{X -243.418,Y 331.859,Z -30.000,A 0.015,B 0.000,C 180.000} C_DIS
LIN {X -392.590,Y 331.856,Z -30.000,A 0.015,B -0.000,C 180.000} C_DIS
CIRC {X -395.315,Y 330.727,Z -30.000,A 0.015,B -0.000,C -180.000},{X -396.443,Y 328.002,Z -30.000,A 0.015,B 0.000,C 180.000} C_DIS
LIN {X -396.436,Y 62.494,Z -30.000,A 0.015,B -0.000,C 180.000} C_DIS
CIRC {X -395.324,Y 60.720,Z -30.000,A 0.015,B -0.000,C 180.000},{X -393.243,Y 60.949,Z -30.000,A 0.015,B -0.000,C -180.000} C_DIS
CIRC {X -391.486,Y 62.347,Z -30.000,A 0.015,B 0.000,C -180.000},{X -389.736,Y 63.754,Z -30.000,A 0.015,B -0.000,C 180.000} C_DIS
CIRC {X -387.852,Y 64.994,Z -30.000,A 0.015,B 0.000,C 180.000},{X -385.763,Y 65.845,Z -30.000,A 0.015,B -0.000,C -180.000} C_DIS
CIRC {X -380.353,Y 67.351,Z -30.000,A 0.015,B -0.000,C -180.000},{X -374.893,Y 68.663,Z -30.000,A 0.015,B -0.000,C 180.000} C_DIS
CIRC {X -369.286,Y 69.312,Z -30.000,A 0.015,B 0.000,C -180.000},{X -363.665,Y 68.807,Z -30.000,A 0.015,B 0.000,C -180.000} C_DIS
CIRC {X -356.428,Y 66.727,Z -30.000,A 0.015,B 0.000,C 180.000},{X -349.667,Y 63.414,Z -30.000,A 0.015,B -0.000,C -180.000} C_DIS
CIRC {X -343.621,Y 58.915,Z -30.000,A 0.015,B -0.000,C 180.000},{X -338.549,Y 53.342,Z -30.000,A 0.015,B 0.000,C -180.000} C_DIS
LIN {X -317.711,Y 18.121,Z -30.000,A 0.015,B 0.000,C 180.000} C_DIS
CIRC {X -314.859,Y 11.626,Z -30.000,A 0.015,B 0.000,C 180.000},{X -313.481,Y 4.668,Z -30.000,A 0.015,B 0.000,C 180.000} C_DIS
CIRC {X -313.222,Y -2.387,Z -30.000,A 0.015,B -0.000,C 180.000},{X -313.667,Y -9.433,Z -30.000,A 0.015,B 0.000,C -180.000} C_DIS
CIRC {X -314.274,Y -12.421,Z -30.000,A 0.015,B -0.000,C -180.000},{X -315.391,Y -15.259,Z -30.000,A 0.015,B -0.000,C 180.000} C_DIS
CIRC {X -316.798,Y -17.952,Z -30.000,A 0.015,B 0.000,C -180.000},{X -318.307,Y -20.590,Z -30.000,A 0.015,B 0.000,C 180.000} C_DIS
CIRC {X -318.332,Y -22.807,Z -30.000,A 0.015,B -0.000,C 180.000},{X -316.416,Y -23.922,Z -30.000,A 0.015,B 0.000,C 180.000} C_DIS
LIN {X -77.125,Y -23.922,Z -30.000,A 0.015,B 0.000,C -180.000} C_DIS
CIRC {X -75.191,Y -22.806,Z -30.000,A 0.015,B 0.000,C 180.000},{X -75.190,Y -20.573,Z -30.000,A 0.015,B 0.000,C -180.000} C_DIS
CIRC {X -78.743,Y -12.558,Z -30.000,A 0.015,B 0.000,C 180.000},{X -80.539,Y -3.975,Z -30.000,A 0.015,B 0.000,C 180.000} C_DIS
CIRC {X -80.321,Y 4.811,Z -30.000,A 0.015,B 0.000,C 180.000},{X -77.929,Y 13.268,Z -30.000,A 0.015,B 0.000,C 180.000} C_DIS
LIN {X -57.473,Y 49.896,Z -30.000,A 0.015,B 0.000,C -180.000} C_DIS
CIRC {X -51.318,Y 57.801,Z -30.000,A 0.015,B 0.000,C -180.000},{X -43.247,Y 63.736,Z -30.000,A 0.015,B 0.000,C -180.000} C_DIS
CIRC {X -34.024,Y 67.545,Z -30.000,A 0.015,B 0.000,C -180.000},{X -24.210,Y 69.350,Z -30.000,A 0.015,B 0.000,C -180.000} C_DIS
CIRC {X -18.883,Y 69.276,Z -30.000,A 0.015,B 0.000,C 180.000},{X -13.657,Y 68.243,Z -30.000,A 0.015,B 0.000,C 180.000} C_DIS
CIRC {X -8.663,Y 66.420,Z -30.000,A 0.015,B 0.000,C -180.000},{X -3.943,Y 63.973,Z -30.000,A 0.015,B 0.000,C 180.000} C_DIS
CIRC {X -2.955,Y 63.299,Z -30.000,A 0.015,B 0.000,C 180.000},{X -2.048,Y 62.519,Z -30.000,A 0.015,B 0.000,C 180.000} C_DIS
CIRC {X -1.169,Y 61.711,Z -30.000,A 0.015,B -0.000,C 180.000},{X -0.255,Y 60.942,Z -30.000,A 0.015,B 0.000,C 180.000} C_DIS
CIRC {X 1.817,Y 60.701,Z -30.000,A 0.015,B -0.000,C 180.000},{X 2.929,Y 62.467,Z -30.000,A 0.015,B 0.000,C -180.000} C_DIS
LIN {X 2.922,Y 328.012,Z -30.000,A 0.015,B -0.000,C -180.000} C_DIS
CIRC {X 1.793,Y 330.737,Z -30.000,A 0.015,B -0.000,C -180.000},{X -0.931,Y 331.865,Z -30.000,A 0.015,B 0.000,C -180.000} C_DIS
LIN {X -150.097,Y 331.861,Z -30.000,A 0.015,B 0.000,C -180.000} C_DIS
CIRC {X -151.729,Y 330.791,Z -30.000,A 0.015,B 0.000,C 180.000},{X -151.400,Y 328.867,Z -30.000,A 0.015,B 0.000,C 180.000} C_DIS
CIRC {X -143.852,Y 317.774,Z -30.000,A 0.015,B 0.000,C 180.000},{X -139.985,Y 304.927,Z -30.000,A 0.015,B -0.000,C 180.000} C_DIS
CIRC {X -140.277,Y 291.494,Z -30.000,A 0.015,B -0.000,C -180.000},{X -144.817,Y 278.849,Z -30.000,A 0.015,B 0.000,C -180.000} C_DIS
CIRC {X -150.766,Y 271.066,Z -30.000,A 0.015,B 0.000,C -180.000},{X -158.707,Y 265.332,Z -30.000,A 0.015,B 0.000,C -180.000} C_DIS
CIRC {X -167.703,Y 261.628,Z -30.000,A 0.015,B 0.000,C 180.000},{X -177.210,Y 259.566,Z -30.000,A 0.015,B 0.000,C -180.000} C_DIS
LIN {X -214.895,Y 259.478,Z -30.000,A 0.015,B 0.000,C -180.000} C_DIS
CIRC {X -224.717,Y 260.809,Z -30.000,A 0.015,B -0.000,C -180.000},{X -233.829,Y 264.708,Z -30.000,A 0.015,B 0.000,C 180.000} C_DIS
CIRC {X -241.728,Y 270.636,Z -30.000,A 0.015,B 0.000,C -180.000},{X -248.219,Y 278.079,Z -30.000,A 0.015,B 0.000,C -180.000} C_DIS
CIRC {X -250.523,Y 282.114,Z -30.000,A 0.015,B 0.000,C 180.000},{X -252.036,Y 286.507,Z -30.000,A 0.015,B -0.000,C 180.000} C_DIS
CIRC {X -253.107,Y 291.008,Z -30.000,A 0.015,B 0.000,C 180.000},{X -254.137,Y 295.519,Z -30.000,A 0.015,B 0.000,C -180.000} C_DIS
CIRC {X -254.543,Y 299.223,Z -30.000,A 0.015,B 0.000,C -180.000},{X -254.124,Y 302.925,Z -30.000,A 0.015,B 0.000,C -180.000} C_DIS
CIRC {X -253.367,Y 306.551,Z -30.000,A 0.015,B 0.000,C -180.000},{X -252.742,Y 310.202,Z -30.000,A 0.015,B 0.000,C -180.000} C_DIS
CIRC {X -251.354,Y 315.362,Z -30.000,A 0.015,B 0.000,C -180.000},{X -248.866,Y 320.092,Z -30.000,A 0.015,B 0.000,C -180.000} C_DIS
CIRC {X -247.388,Y 322.211,Z -30.000,A 0.015,B 0.000,C 180.000},{X -245.853,Y 324.289,Z -30.000,A 0.015,B 0.000,C 180.000} C_DIS
LIN {X -245.681,Y 324.893,Z -29.830,A 0.015,B 0.000,C 180.000} C_DIS
LIN {X -245.752,Y 325.350,Z -29.365,A 0.015,B -0.000,C 180.000} C_DIS
LIN {X -245.819,Y 325.506,Z -28.730,A 0.015,B 0.000,C 180.000} C_DIS
$VEL.CP = 1.00000
LIN {X -245.819,Y 325.506,Z 11.000,A 0.015,B 0.000,C 180.000} C_DIS
$VEL.CP = 1.00000
LIN {X -398.500,Y 339.199,Z 11.000,A 0.015,B 0.000,C -180.000} C_DIS
$VEL.CP = 0.10000
LIN {X -398.500,Y 339.199,Z -8.231,A 0.015,B 0.000,C -180.000} C_DIS
LIN {X -398.507,Y 339.199,Z -8.362,A 0.015,B -0.000,C -180.000} C_DIS
LIN {X -398.770,Y 339.192,Z -9.014,A 0.015,B 0.000,C -180.000} C_DIS
LIN {X -399.336,Y 339.133,Z -9.426,A 0.015,B 0.000,C -180.000} C_DIS
LIN {X -399.692,Y 339.076,Z -9.499,A 0.015,B 0.000,C -180.000} C_DIS
LIN {X -399.717,Y 339.072,Z -9.500,A 0.015,B 0.000,C -180.000} C_DIS
LIN {X -400.552,Y 338.848,Z -9.530,A 0.015,B 0.000,C -180.000} C_DIS
LIN {X -400.596,Y 338.832,Z -9.532,A 0.015,B 0.000,C 180.000} C_DIS
LIN {X -401.281,Y 338.494,Z -9.559,A 0.015,B -0.000,C -180.000} C_DIS
LIN {X -401.404,Y 338.418,Z -9.564,A 0.015,B -0.000,C 180.000} C_DIS
LIN {X -402.842,Y 337.053,Z -9.633,A 0.015,B -0.000,C -180.000} C_DIS
LIN {X -402.866,Y 337.018,Z -9.635,A 0.015,B -0.000,C -180.000} C_DIS
LIN {X -403.753,Y 334.430,Z -9.732,A 0.015,B 0.000,C 180.000} C_DIS
LIN {X -403.779,Y 333.946,Z -9.749,A 0.015,B -0.000,C 180.000} C_DIS
LIN {X -403.787,Y 333.653,Z -9.759,A 0.015,B -0.000,C -180.000} C_DIS
LIN {X -403.787,Y 333.050,Z -9.780,A 0.015,B 0.000,C -180.000} C_DIS
LIN {X -401.252,Y 328.076,Z -9.982,A 0.015,B 0.000,C 180.000} C_DIS
LIN {X -395.738,Y 327.203,Z -10.185,A 0.015,B 0.000,C -180.000} C_DIS
LIN {X -391.790,Y 331.150,Z -10.387,A 0.015,B -0.000,C 180.000} C_DIS
LIN {X -392.664,Y 336.664,Z -10.589,A 0.015,B -0.000,C -180.000} C_DIS
LIN {X -397.638,Y 339.199,Z -10.792,A 0.015,B -0.000,C 180.000} C_DIS
LIN {X -398.507,Y 339.199,Z -10.822,A 0.015,B 0.000,C -180.000} C_DIS
LIN {X -399.336,Y 339.133,Z -10.851,A 0.015,B -0.000,C -180.000} C_DIS
LIN {X -399.692,Y 339.076,Z -10.864,A 0.015,B -0.000,C -180.000} C_DIS
LIN {X -400.552,Y 338.848,Z -10.895,A 0.015,B 0.000,C 180.000} C_DIS
LIN {X -400.596,Y 338.832,Z -10.896,A 0.015,B 0.000,C -180.000} C_DIS
LIN {X -401.281,Y 338.494,Z -10.923,A 0.015,B -0.000,C -180.000} C_DIS
LIN {X -401.404,Y 338.418,Z -10.928,A 0.015,B -0.000,C -180.000} C_DIS
LIN {X -402.842,Y 337.053,Z -10.998,A 0.015,B -0.000,C -180.000} C_DIS
LIN {X -402.866,Y 337.018,Z -10.999,A 0.015,B -0.000,C -180.000} C_DIS
LIN {X -403.753,Y 334.430,Z -11.096,A 0.015,B 0.000,C -180.000} C_DIS
LIN {X -403.779,Y 333.946,Z -11.113,A 0.015,B 0.000,C -180.000} C_DIS
LIN {X -403.787,Y 333.653,Z -11.123,A 0.015,B 0.000,C -180.000} C_DIS
LIN {X -403.787,Y 333.050,Z -11.144,A 0.015,B -0.000,C -180.000} C_DIS
LIN {X -401.252,Y 328.076,Z -11.347,A 0.015,B 0.000,C 180.000} C_DIS
LIN {X -395.738,Y 327.203,Z -11.549,A 0.015,B -0.000,C 180.000} C_DIS
LIN {X -391.790,Y 331.150,Z -11.751,A 0.015,B -0.000,C 180.000} C_DIS
LIN {X -392.664,Y 336.664,Z -11.954,A 0.015,B 0.000,C -180.000} C_DIS
LIN {X -397.638,Y 339.199,Z -12.156,A 0.015,B 0.000,C -180.000} C_DIS
LIN {X -398.507,Y 339.199,Z -12.187,A 0.015,B -0.000,C -180.000} C_DIS
LIN {X -399.336,Y 339.133,Z -12.216,A 0.015,B 0.000,C 180.000} C_DIS
LIN {X -399.692,Y 339.076,Z -12.228,A 0.015,B 0.000,C -180.000} C_DIS
LIN {X -400.552,Y 338.848,Z -12.259,A 0.015,B 0.000,C -180.000} C_DIS
LIN {X -400.596,Y 338.832,Z -12.261,A 0.015,B -0.000,C 180.000} C_DIS
LIN {X -401.281,Y 338.494,Z -12.288,A 0.015,B -0.000,C -180.000} C_DIS
LIN {X -401.404,Y 338.418,Z -12.293,A 0.015,B 0.000,C -180.000} C_DIS
LIN {X -402.842,Y 337.053,Z -12.362,A 0.015,B 0.000,C -180.000} C_DIS
LIN {X -402.866,Y 337.018,Z -12.364,A 0.015,B 0.000,C 180.000} C_DIS
LIN {X -403.753,Y 334.430,Z -12.461,A 0.015,B -0.000,C -180.000} C_DIS
LIN {X -403.779,Y 333.946,Z -12.478,A 0.015,B 0.000,C -180.000} C_DIS
LIN {X -403.787,Y 333.653,Z -12.488,A 0.015,B -0.000,C 180.000} C_DIS
LIN {X -403.787,Y 333.050,Z -12.509,A 0.015,B 0.000,C -180.000} C_DIS
LIN {X -401.252,Y 328.076,Z -12.711,A 0.015,B 0.000,C 180.000} C_DIS
LIN {X -395.738,Y 327.203,Z -12.914,A 0.015,B -0.000,C 180.000} C_DIS
LIN {X -391.790,Y 331.150,Z -13.116,A 0.015,B -0.000,C 180.000} C_DIS
LIN {X -392.664,Y 336.664,Z -13.318,A 0.015,B 0.000,C -180.000} C_DIS
LIN {X -397.638,Y 339.199,Z -13.521,A 0.015,B 0.000,C -180.000} C_DIS
LIN {X -398.507,Y 339.199,Z -13.551,A 0.015,B -0.000,C 180.000} C_DIS
LIN {X -399.336,Y 339.133,Z -13.580,A 0.015,B 0.000,C -180.000} C_DIS
LIN {X -399.692,Y 339.076,Z -13.593,A 0.015,B 0.000,C -180.000} C_DIS
LIN {X -400.552,Y 338.848,Z -13.624,A 0.015,B -0.000,C 180.000} C_DIS
LIN {X -400.596,Y 338.832,Z -13.625,A 0.015,B -0.000,C -180.000} C_DIS
LIN {X -401.281,Y 338.494,Z -13.652,A 0.015,B -0.000,C 180.000} C_DIS
LIN {X -401.404,Y 338.418,Z -13.657,A 0.015,B 0.000,C 180.000} C_DIS
LIN {X -402.842,Y 337.053,Z -13.727,A 0.015,B -0.000,C -180.000} C_DIS
LIN {X -402.866,Y 337.018,Z -13.728,A 0.015,B -0.000,C -180.000} C_DIS
LIN {X -403.753,Y 334.430,Z -13.825,A 0.015,B 0.000,C -180.000} C_DIS
LIN {X -403.779,Y 333.946,Z -13.842,A 0.015,B -0.000,C -180.000} C_DIS
LIN {X -403.787,Y 333.653,Z -13.852,A 0.015,B 0.000,C 180.000} C_DIS
LIN {X -403.787,Y 333.050,Z -13.873,A 0.015,B -0.000,C -180.000} C_DIS
LIN {X -401.252,Y 328.076,Z -14.076,A 0.015,B -0.000,C 180.000} C_DIS
LIN {X -395.738,Y 327.203,Z -14.278,A 0.015,B -0.000,C 180.000} C_DIS
LIN {X -391.790,Y 331.150,Z -14.481,A 0.015,B -0.000,C -180.000} C_DIS
LIN {X -392.664,Y 336.664,Z -14.683,A 0.015,B -0.000,C -180.000} C_DIS
LIN {X -397.638,Y 339.199,Z -14.885,A 0.015,B -0.000,C 180.000} C_DIS
LIN {X -398.507,Y 339.199,Z -14.916,A 0.015,B -0.000,C -180.000} C_DIS
LIN {X -399.336,Y 339.133,Z -14.945,A 0.015,B 0.000,C 180.000} C_DIS
LIN {X -399.692,Y 339.076,Z -14.957,A 0.015,B 0.000,C -180.000} C_DIS
LIN {X -400.552,Y 338.848,Z -14.988,A 0.015,B 0.000,C 180.000} C_DIS
LIN {X -400.596,Y 338.832,Z -14.990,A 0.015,B 0.000,C -180.000} C_DIS
LIN {X -401.281,Y 338.494,Z -15.017,A 0.015,B -0.000,C -180.000} C_DIS
LIN {X -401.404,Y 338.418,Z -15.022,A 0.015,B 0.000,C -180.000} C_DIS
LIN {X -402.842,Y 337.053,Z -15.092,A 0.015,B -0.000,C -180.000} C_DIS
LIN {X -402.866,Y 337.018,Z -15.093,A 0.015,B -0.000,C 180.000} C_DIS
LIN {X -403.753,Y 334.430,Z -15.190,A 0.015,B 0.000,C -180.000} C_DIS
LIN {X -403.779,Y 333.946,Z -15.207,A 0.015,B 0.000,C 180.000} C_DIS
LIN {X -403.787,Y 333.653,Z -15.217,A 0.015,B -0.000,C -180.000} C_DIS
LIN {X -403.787,Y 333.050,Z -15.238,A 0.015,B -0.000,C -180.000} C_DIS
LIN {X -401.252,Y 328.076,Z -15.440,A 0.015,B 0.000,C -180.000} C_DIS
LIN {X -395.738,Y 327.203,Z -15.643,A 0.015,B 0.000,C 180.000} C_DIS
LIN {X -391.790,Y 331.150,Z -15.845,A 0.015,B -0.000,C -180.000} C_DIS
LIN {X -392.664,Y 336.664,Z -16.047,A 0.015,B -0.000,C -180.000} C_DIS
LIN {X -397.638,Y 339.199,Z -16.250,A 0.015,B -0.000,C -180.000} C_DIS
LIN {X -398.507,Y 339.199,Z -16.280,A 0.015,B -0.000,C -180.000} C_DIS
LIN {X -399.336,Y 339.133,Z -16.309,A 0.015,B 0.000,C 180.000} C_DIS
LIN {X -399.692,Y 339.076,Z -16.322,A 0.015,B 0.000,C -180.000} C_DIS
LIN {X -400.552,Y 338.848,Z -16.353,A 0.015,B 0.000,C 180.000} C_DIS
LIN {X -400.596,Y 338.832,Z -16.355,A 0.015,B 0.000,C 180.000} C_DIS
LIN {X -401.281,Y 338.494,Z -16.381,A 0.015,B -0.000,C -180.000} C_DIS
LIN {X -401.404,Y 338.418,Z -16.386,A 0.015,B 0.000,C -180.000} C_DIS
LIN {X -402.842,Y 337.053,Z -16.456,A 0.015,B 0.000,C 180.000} C_DIS
LIN {X -402.866,Y 337.018,Z -16.458,A 0.015,B -0.000,C 180.000} C_DIS
LIN {X -403.753,Y 334.430,Z -16.554,A 0.015,B -0.000,C 180.000} C_DIS
LIN {X -403.779,Y 333.946,Z -16.571,A 0.015,B 0.000,C 180.000} C_DIS
LIN {X -403.787,Y 333.653,Z -16.581,A 0.015,B 0.000,C -180.000} C_DIS
LIN {X -403.787,Y 333.050,Z -16.603,A 0.015,B 0.000,C 180.000} C_DIS
LIN {X -401.252,Y 328.076,Z -16.805,A 0.015,B 0.000,C 180.000} C_DIS
LIN {X -395.738,Y 327.203,Z -17.007,A 0.015,B 0.000,C -180.000} C_DIS
LIN {X -391.790,Y 331.150,Z -17.210,A 0.015,B 0.000,C -180.000} C_DIS
LIN {X -392.664,Y 336.664,Z -17.412,A 0.015,B 0.000,C 180.000} C_DIS
LIN {X -397.638,Y 339.199,Z -17.614,A 0.015,B -0.000,C -180.000} C_DIS
LIN {X -398.507,Y 339.199,Z -17.645,A 0.015,B 0.000,C 180.000} C_DIS
LIN {X -399.336,Y 339.133,Z -17.674,A 0.015,B -0.000,C -180.000} C_DIS
LIN {X -399.692,Y 339.076,Z -17.686,A 0.015,B -0.000,C -180.000} C_DIS
LIN {X -400.552,Y 338.848,Z -17.718,A 0.015,B 0.000,C -180.000} C_DIS
LIN {X -400.596,Y 338.832,Z -17.719,A 0.015,B -0.000,C -180.000} C_DIS
LIN {X -401.281,Y 338.494,Z -17.746,A 0.015,B 0.000,C -180.000} C_DIS
LIN {X -401.404,Y 338.418,Z -17.751,A 0.015,B -0.000,C -180.000} C_DIS
LIN {X -402.842,Y 337.053,Z -17.821,A 0.015,B 0.000,C 180.000} C_DIS
LIN {X -402.866,Y 337.018,Z -17.822,A 0.015,B 0.000,C -180.000} C_DIS
LIN {X -403.753,Y 334.430,Z -17.919,A 0.015,B 0.000,C -180.000} C_DIS
LIN {X -403.779,Y 333.946,Z -17.936,A 0.015,B 0.000,C 180.000} C_DIS
LIN {X -403.787,Y 333.653,Z -17.946,A 0.015,B 0.000,C -180.000} C_DIS
LIN {X -403.787,Y 333.050,Z -17.967,A 0.015,B 0.000,C 180.000} C_DIS
LIN {X -401.252,Y 328.076,Z -18.169,A 0.015,B 0.000,C 180.000} C_DIS
LIN {X -395.738,Y 327.203,Z -18.372,A 0.015,B -0.000,C -180.000} C_DIS
LIN {X -391.790,Y 331.150,Z -18.574,A 0.015,B 0.000,C -180.000} C_DIS
LIN {X -392.664,Y 336.664,Z -18.777,A 0.015,B 0.000,C -180.000} C_DIS
LIN {X -397.638,Y 339.199,Z -18.979,A 0.015,B -0.000,C -180.000} C_DIS
LIN {X -398.507,Y 339.199,Z -19.009,A 0.015,B 0.000,C -180.000} C_DIS
LIN {X -399.336,Y 339.133,Z -19.038,A 0.015,B 0.000,C 180.000} C_DIS
LIN {X -399.692,Y 339.076,Z -19.051,A 0.015,B 0.000,C 180.000} C_DIS
LIN {X -400.552,Y 338.848,Z -19.082,A 0.015,B 0.000,C -180.000} C_DIS
LIN {X -400.596,Y 338.832,Z -19.084,A 0.015,B -0.000,C -180.000} C_DIS
LIN {X -401.281,Y 338.494,Z -19.110,A 0.015,B 0.000,C -180.000} C_DIS
LIN {X -401.404,Y 338.418,Z -19.115,A 0.015,B -0.000,C 180.000} C_DIS
LIN {X -402.842,Y 337.053,Z -19.185,A 0.015,B -0.000,C -180.000} C_DIS
LIN {X -402.866,Y 337.018,Z -19.187,A 0.015,B 0.000,C 180.000} C_DIS
LIN {X -403.753,Y 334.430,Z -19.283,A 0.015,B -0.000,C 180.000} C_DIS
LIN {X -403.779,Y 333.946,Z -19.300,A 0.015,B 0.000,C 180.000} C_DIS
LIN {X -403.787,Y 333.653,Z -19.311,A 0.015,B 0.000,C -180.000} C_DIS
LIN {X -403.787,Y 333.050,Z -19.332,A 0.015,B -0.000,C -180.000} C_DIS
LIN {X -401.252,Y 328.076,Z -19.534,A 0.015,B 0.000,C -180.000} C_DIS
LIN {X -395.738,Y 327.203,Z -19.736,A 0.015,B -0.000,C 180.000} C_DIS
LIN {X -391.790,Y 331.150,Z -19.939,A 0.015,B -0.000,C 180.000} C_DIS
LIN {X -392.664,Y 336.664,Z -20.141,A 0.015,B -0.000,C 180.000} C_DIS
LIN {X -397.638,Y 339.199,Z -20.343,A 0.015,B -0.000,C -180.000} C_DIS
LIN {X -398.507,Y 339.199,Z -20.374,A 0.015,B 0.000,C 180.000} C_DIS
LIN {X -399.336,Y 339.133,Z -20.403,A 0.015,B 0.000,C 180.000} C_DIS
LIN {X -399.692,Y 339.076,Z -20.415,A 0.015,B -0.000,C -180.000} C_DIS
LIN {X -400.552,Y 338.848,Z -20.447,A 0.015,B -0.000,C 180.000} C_DIS
LIN {X -400.596,Y 338.832,Z -20.448,A 0.015,B 0.000,C -180.000} C_DIS
LIN {X -401.281,Y 338.494,Z -20.475,A 0.015,B 0.000,C 180.000} C_DIS
LIN {X -401.404,Y 338.418,Z -20.480,A 0.015,B -0.000,C -180.000} C_DIS
LIN {X -402.842,Y 337.053,Z -20.550,A 0.015,B 0.000,C -180.000} C_DIS
LIN {X -402.866,Y 337.018,Z -20.551,A 0.015,B -0.000,C -180.000} C_DIS
LIN {X -403.753,Y 334.430,Z -20.648,A 0.015,B 0.000,C -180.000} C_DIS
LIN {X -403.779,Y 333.946,Z -20.665,A 0.015,B -0.000,C -180.000} C_DIS
LIN {X -403.787,Y 333.653,Z -20.675,A 0.015,B -0.000,C -180.000} C_DIS
LIN {X -403.787,Y 333.050,Z -20.696,A 0.015,B 0.000,C -180.000} C_DIS
LIN {X -401.252,Y 328.076,Z -20.899,A 0.015,B 0.000,C 180.000} C_DIS
LIN {X -395.738,Y 327.203,Z -21.101,A 0.015,B 0.000,C -180.000} C_DIS
LIN {X -391.790,Y 331.150,Z -21.303,A 0.015,B 0.000,C -180.000} C_DIS
LIN {X -392.664,Y 336.664,Z -21.506,A 0.015,B 0.000,C -180.000} C_DIS
LIN {X -397.638,Y 339.199,Z -21.708,A 0.015,B 0.000,C 180.000} C_DIS
LIN {X -398.507,Y 339.199,Z -21.738,A 0.015,B -0.000,C -180.000} C_DIS
LIN {X -399.336,Y 339.133,Z -21.767,A 0.015,B -0.000,C -180.000} C_DIS
LIN {X -399.692,Y 339.076,Z -21.780,A 0.015,B 0.000,C 180.000} C_DIS
LIN {X -400.552,Y 338.848,Z -21.811,A 0.015,B -0.000,C 180.000} C_DIS
LIN {X -400.596,Y 338.832,Z -21.813,A 0.015,B -0.000,C 180.000} C_DIS
LIN {X -401.281,Y 338.494,Z -21.839,A 0.015,B 0.000,C 180.000} C_DIS
LIN {X -401.404,Y 338.418,Z -21.845,A 0.015,B 0.000,C 180.000} C_DIS
LIN {X -402.842,Y 337.053,Z -21.914,A 0.015,B -0.000,C -180.000} C_DIS
LIN {X -402.866,Y 337.018,Z -21.916,A 0.015,B 0.000,C 180.000} C_DIS
LIN {X -403.753,Y 334.430,Z -22.012,A 0.015,B 0.000,C -180.000} C_DIS
LIN {X -403.779,Y 333.946,Z -22.029,A 0.015,B 0.000,C 180.000} C_DIS
LIN {X -403.787,Y 333.653,Z -22.040,A 0.015,B 0.000,C 180.000} C_DIS
LIN {X -403.787,Y 333.050,Z -22.061,A 0.015,B 0.000,C -180.000} C_DIS
LIN {X -401.252,Y 328.076,Z -22.263,A 0.015,B 0.000,C -180.000} C_DIS
LIN {X -395.738,Y 327.203,Z -22.465,A 0.015,B -0.000,C -180.000} C_DIS
LIN {X -391.790,Y 331.150,Z -22.668,A 0.015,B -0.000,C -180.000} C_DIS
LIN {X -392.664,Y 336.664,Z -22.870,A 0.015,B -0.000,C 180.000} C_DIS
LIN {X -397.638,Y 339.199,Z -23.073,A 0.015,B 0.000,C -180.000} C_DIS
LIN {X -398.507,Y 339.199,Z -23.103,A 0.015,B -0.000,C -180.000} C_DIS
LIN {X -399.336,Y 339.133,Z -23.132,A 0.015,B 0.000,C 180.000} C_DIS
LIN {X -399.692,Y 339.076,Z -23.145,A 0.015,B 0.000,C 180.000} C_DIS
LIN {X -400.552,Y 338.848,Z -23.176,A 0.015,B 0.000,C 180.000} C_DIS
LIN {X -400.596,Y 338.832,Z -23.177,A 0.015,B -0.000,C 180.000} C_DIS
LIN {X -401.281,Y 338.494,Z -23.204,A 0.015,B 0.000,C -180.000} C_DIS
LIN {X -401.404,Y 338.418,Z -23.209,A 0.015,B 0.000,C -180.000} C_DIS
LIN {X -402.842,Y 337.053,Z -23.279,A 0.015,B -0.000,C -180.000} C_DIS
LIN {X -402.866,Y 337.018,Z -23.280,A 0.015,B 0.000,C 180.000} C_DIS
LIN {X -403.753,Y 334.430,Z -23.377,A 0.015,B -0.000,C 180.000} C_DIS
LIN {X -403.779,Y 333.946,Z -23.394,A 0.015,B 0.000,C 180.000} C_DIS
LIN {X -403.787,Y 333.653,Z -23.404,A 0.015,B 0.000,C 180.000} C_DIS
LIN {X -403.787,Y 333.050,Z -23.425,A 0.015,B -0.000,C -180.000} C_DIS
LIN {X -401.252,Y 328.076,Z -23.628,A 0.015,B -0.000,C -180.000} C_DIS
LIN {X -395.738,Y 327.203,Z -23.830,A 0.015,B -0.000,C -180.000} C_DIS
LIN {X -391.790,Y 331.150,Z -24.032,A 0.015,B 0.000,C -180.000} C_DIS
LIN {X -392.664,Y 336.664,Z -24.235,A 0.015,B 0.000,C -180.000} C_DIS
LIN {X -397.638,Y 339.199,Z -24.437,A 0.015,B -0.000,C -180.000} C_DIS
LIN {X -398.507,Y 339.199,Z -24.467,A 0.015,B -0.000,C -180.000} C_DIS
LIN {X -399.336,Y 339.133,Z -24.496,A 0.015,B 0.000,C 180.000} C_DIS
LIN {X -399.692,Y 339.076,Z -24.509,A 0.015,B -0.000,C 180.000} C_DIS
LIN {X -400.552,Y 338.848,Z -24.540,A 0.015,B -0.000,C 180.000} C_DIS
LIN {X -400.596,Y 338.832,Z -24.542,A 0.015,B 0.000,C 180.000} C_DIS
LIN {X -401.281,Y 338.494,Z -24.569,A 0.015,B -0.000,C -180.000} C_DIS
LIN {X -401.404,Y 338.418,Z -24.574,A 0.015,B -0.000,C -180.000} C_DIS
LIN {X -402.842,Y 337.053,Z -24.643,A 0.015,B 0.000,C 180.000} C_DIS
LIN {X -402.866,Y 337.018,Z -24.645,A 0.015,B -0.000,C -180.000} C_DIS
LIN {X -403.753,Y 334.430,Z -24.742,A 0.015,B 0.000,C -180.000} C_DIS
LIN {X -403.779,Y 333.946,Z -24.758,A 0.015,B 0.000,C -180.000} C_DIS
LIN {X -403.787,Y 333.653,Z -24.769,A 0.015,B 0.000,C -180.000} C_DIS
LIN {X -403.787,Y 333.050,Z -24.790,A 0.015,B 0.000,C -180.000} C_DIS
LIN {X -401.252,Y 328.076,Z -24.992,A 0.015,B 0.000,C -180.000} C_DIS
LIN {X -395.738,Y 327.203,Z -25.195,A 0.015,B 0.000,C 180.000} C_DIS
LIN {X -391.790,Y 331.150,Z -25.397,A 0.015,B 0.000,C 180.000} C_DIS
LIN {X -392.664,Y 336.664,Z -25.599,A 0.015,B -0.000,C -180.000} C_DIS
LIN {X -397.638,Y 339.199,Z -25.802,A 0.015,B -0.000,C -180.000} C_DIS
LIN {X -398.507,Y 339.199,Z -25.832,A 0.015,B -0.000,C -180.000} C_DIS
LIN {X -399.336,Y 339.133,Z -25.861,A 0.015,B -0.000,C -180.000} C_DIS
LIN {X -399.692,Y 339.076,Z -25.874,A 0.015,B 0.000,C 180.000} C_DIS
LIN {X -400.552,Y 338.848,Z -25.905,A 0.015,B 0.000,C -180.000} C_DIS
LIN {X -400.596,Y 338.832,Z -25.906,A 0.015,B -0.000,C -180.000} C_DIS
LIN {X -401.281,Y 338.494,Z -25.933,A 0.015,B 0.000,C 180.000} C_DIS
LIN {X -401.404,Y 338.418,Z -25.938,A 0.015,B 0.000,C -180.000} C_DIS
LIN {X -402.842,Y 337.053,Z -26.008,A 0.015,B 0.000,C 180.000} C_DIS
LIN {X -402.866,Y 337.018,Z -26.009,A 0.015,B 0.000,C 180.000} C_DIS
LIN {X -403.753,Y 334.430,Z -26.106,A 0.015,B 0.000,C -180.000} C_DIS
LIN {X -403.779,Y 333.946,Z -26.123,A 0.015,B 0.000,C 180.000} C_DIS
LIN {X -403.787,Y 333.653,Z -26.133,A 0.015,B 0.000,C -180.000} C_DIS
LIN {X -403.787,Y 333.050,Z -26.154,A 0.015,B 0.000,C -180.000} C_DIS
LIN {X -401.252,Y 328.076,Z -26.357,A 0.015,B 0.000,C 180.000} C_DIS
LIN {X -395.738,Y 327.203,Z -26.559,A 0.015,B 0.000,C -180.000} C_DIS
LIN {X -391.790,Y 331.150,Z -26.761,A 0.015,B 0.000,C 180.000} C_DIS
LIN {X -392.664,Y 336.664,Z -26.964,A 0.015,B -0.000,C 180.000} C_DIS
LIN {X -397.638,Y 339.199,Z -27.166,A 0.015,B 0.000,C -180.000} C_DIS
LIN {X -398.507,Y 339.199,Z -27.196,A 0.015,B -0.000,C -180.000} C_DIS
LIN {X -399.336,Y 339.133,Z -27.226,A 0.015,B -0.000,C -180.000} C_DIS
LIN {X -399.692,Y 339.076,Z -27.238,A 0.015,B 0.000,C -180.000} C_DIS
LIN {X -400.552,Y 338.848,Z -27.269,A 0.015,B 0.000,C -180.000} C_DIS
LIN {X -400.596,Y 338.832,Z -27.271,A 0.015,B 0.000,C -180.000} C_DIS
LIN {X -401.281,Y 338.494,Z -27.298,A 0.015,B 0.000,C -180.000} C_DIS
LIN {X -401.404,Y 338.418,Z -27.303,A 0.015,B 0.000,C -180.000} C_DIS
LIN {X -402.842,Y 337.053,Z -27.372,A 0.015,B -0.000,C 180.000} C_DIS
LIN {X -402.866,Y 337.018,Z -27.374,A 0.015,B 0.000,C -180.000} C_DIS
LIN {X -403.753,Y 334.430,Z -27.471,A 0.015,B 0.000,C 180.000} C_DIS
LIN {X -403.779,Y 333.946,Z -27.488,A 0.015,B 0.000,C -180.000} C_DIS
LIN {X -403.787,Y 333.653,Z -27.498,A 0.015,B 0.000,C -180.000} C_DIS
LIN {X -403.787,Y 333.050,Z -27.519,A 0.015,B 0.000,C 180.000} C_DIS
LIN {X -401.252,Y 328.076,Z -27.721,A 0.015,B 0.000,C -180.000} C_DIS
LIN {X -395.738,Y 327.203,Z -27.924,A 0.015,B -0.000,C -180.000} C_DIS
LIN {X -391.790,Y 331.150,Z -28.126,A 0.015,B 0.000,C -180.000} C_DIS
LIN {X -392.664,Y 336.664,Z -28.328,A 0.015,B 0.000,C 180.000} C_DIS
LIN {X -397.638,Y 339.199,Z -28.531,A 0.015,B -0.000,C -180.000} C_DIS
LIN {X -398.507,Y 339.199,Z -28.561,A 0.015,B -0.000,C 180.000} C_DIS
LIN {X -399.336,Y 339.133,Z -28.590,A 0.015,B -0.000,C -180.000} C_DIS
LIN {X -399.692,Y 339.076,Z -28.603,A 0.015,B 0.000,C 180.000} C_DIS
LIN {X -400.552,Y 338.848,Z -28.634,A 0.015,B -0.000,C 180.000} C_DIS
LIN {X -400.596,Y 338.832,Z -28.635,A 0.015,B 0.000,C 180.000} C_DIS
LIN {X -401.281,Y 338.494,Z -28.662,A 0.015,B 0.000,C -180.000} C_DIS
LIN {X -401.404,Y 338.418,Z -28.667,A 0.015,B -0.000,C -180.000} C_DIS
LIN {X -402.842,Y 337.053,Z -28.737,A 0.015,B -0.000,C 180.000} C_DIS
LIN {X -402.866,Y 337.018,Z -28.738,A 0.015,B 0.000,C -180.000} C_DIS
LIN {X -403.753,Y 334.430,Z -28.835,A 0.015,B 0.000,C 180.000} C_DIS
LIN {X -403.779,Y 333.946,Z -28.852,A 0.015,B 0.000,C 180.000} C_DIS
LIN {X -403.787,Y 333.653,Z -28.862,A 0.015,B 0.000,C 180.000} C_DIS
LIN {X -403.787,Y 333.050,Z -28.883,A 0.015,B -0.000,C -180.000} C_DIS
LIN {X -401.252,Y 328.076,Z -29.086,A 0.015,B -0.000,C 180.000} C_DIS
LIN {X -395.738,Y 327.203,Z -29.288,A 0.015,B -0.000,C 180.000} C_DIS
LIN {X -391.790,Y 331.150,Z -29.491,A 0.015,B 0.000,C -180.000} C_DIS
LIN {X -392.664,Y 336.664,Z -29.693,A 0.015,B 0.000,C -180.000} C_DIS
LIN {X -397.638,Y 339.199,Z -29.895,A 0.015,B 0.000,C -180.000} C_DIS
LIN {X -398.507,Y 339.199,Z -29.926,A 0.015,B 0.000,C 180.000} C_DIS
LIN {X -399.336,Y 339.133,Z -29.955,A 0.015,B 0.000,C -180.000} C_DIS
LIN {X -399.692,Y 339.076,Z -29.967,A 0.015,B -0.000,C 180.000} C_DIS
LIN {X -400.552,Y 338.848,Z -29.998,A 0.015,B 0.000,C 180.000} C_DIS
LIN {X -400.596,Y 338.832,Z -30.000,A 0.015,B 0.000,C 180.000} C_DIS
LIN {X -400.134,Y 339.006,Z -30.000,A 0.015,B 0.000,C -180.000} C_DIS
LIN {X -398.924,Y 339.199,Z -30.000,A 0.015,B 0.000,C 180.000} C_DIS
LIN {X -213.263,Y 339.203,Z -30.000,A 0.015,B 0.000,C -180.000} C_DIS
LIN {X -213.586,Y 339.155,Z -30.000,A 0.015,B 0.000,C -180.000} C_DIS
LIN {X -214.125,Y 339.028,Z -30.000,A 0.015,B -0.000,C -180.000} C_DIS
LIN {X -215.213,Y 338.675,Z -30.000,A 0.015,B 0.000,C 180.000} C_DIS
LIN {X -215.662,Y 338.493,Z -30.000,A 0.015,B 0.000,C 180.000} C_DIS
LIN {X -226.546,Y 333.142,Z -30.000,A 0.015,B 0.000,C 180.000} C_DIS
LIN {X -227.087,Y 332.809,Z -30.000,A 0.015,B 0.000,C -180.000} C_DIS
LIN {X -228.176,Y 331.990,Z -30.000,A 0.015,B 0.000,C 180.000} C_DIS
LIN {X -228.474,Y 331.737,Z -30.000,A 0.015,B 0.000,C 180.000} C_DIS
LIN {X -236.596,Y 324.006,Z -30.000,A 0.015,B 0.000,C -180.000} C_DIS
LIN {X -236.834,Y 323.755,Z -30.000,A 0.015,B -0.000,C 180.000} C_DIS
LIN {X -237.766,Y 322.667,Z -30.000,A 0.015,B 0.000,C 180.000} C_DIS
LIN {X -238.117,Y 322.172,Z -30.000,A 0.015,B -0.000,C -180.000} C_DIS
LIN {X -240.445,Y 318.182,Z -30.000,A 0.015,B -0.000,C -180.000} C_DIS
LIN {X -240.500,Y 318.085,Z -30.000,A 0.015,B -0.000,C -180.000} C_DIS
LIN {X -244.026,Y 311.555,Z -30.000,A 0.015,B 0.000,C -180.000} C_DIS
LIN {X -244.210,Y 311.152,Z -30.000,A 0.015,B 0.000,C -180.000} C_DIS
LIN {X -244.763,Y 309.701,Z -30.000,A 0.015,B -0.000,C 180.000} C_DIS
LIN {X -244.946,Y 309.009,Z -30.000,A 0.015,B 0.000,C 180.000} C_DIS
LIN {X -246.389,Y 299.577,Z -30.000,A 0.015,B 0.000,C -180.000} C_DIS
LIN {X -246.415,Y 299.356,Z -30.000,A 0.015,B 0.000,C -180.000} C_DIS
LIN {X -246.509,Y 298.268,Z -30.000,A 0.015,B 0.000,C 180.000} C_DIS
CIRC {X -246.514,Y 297.751,Z -30.000,A 0.015,B 0.000,C -180.000},{X -246.440,Y 297.239,Z -30.000,A 0.015,B 0.000,C 180.000} C_DIS
LIN {X -245.042,Y 290.986,Z -30.000,A 0.015,B 0.000,C 180.000} C_DIS
LIN {X -245.026,Y 290.918,Z -30.000,A 0.015,B 0.000,C -180.000} C_DIS
LIN {X -244.069,Y 287.015,Z -30.000,A 0.015,B 0.000,C 180.000} C_DIS
LIN {X -243.751,Y 286.197,Z -30.000,A 0.015,B 0.000,C 180.000} C_DIS
LIN {X -241.964,Y 282.932,Z -30.000,A 0.015,B 0.000,C -180.000} C_DIS
LIN {X -241.765,Y 282.612,Z -30.000,A 0.015,B -0.000,C -180.000} C_DIS
LIN {X -239.727,Y 279.710,Z -30.000,A 0.015,B 0.000,C -180.000} C_DIS
LIN {X -239.536,Y 279.464,Z -30.000,A 0.015,B 0.000,C -180.000} C_DIS
LIN {X -237.071,Y 276.562,Z -30.000,A 0.015,B 0.000,C -180.000} C_DIS
LIN {X -236.532,Y 276.053,Z -30.000,A 0.015,B 0.000,C -180.000} C_DIS
LIN {X -232.689,Y 273.151,Z -30.000,A 0.015,B 0.000,C -180.000} C_DIS
LIN {X -232.491,Y 273.012,Z -30.000,A 0.015,B 0.000,C 180.000} C_DIS
LIN {X -229.795,Y 271.265,Z -30.000,A 0.015,B -0.000,C 180.000} C_DIS
LIN {X -229.472,Y 271.079,Z -30.000,A 0.015,B 0.000,C 180.000} C_DIS
LIN {X -227.168,Y 269.924,Z -30.000,A 0.015,B 0.000,C -180.000} C_DIS
LIN {X -226.755,Y 269.750,Z -30.000,A 0.015,B 0.000,C -180.000} C_DIS
LIN {X -223.979,Y 268.793,Z -30.000,A 0.015,B 0.000,C 180.000} C_DIS
LIN {X -223.479,Y 268.663,Z -30.000,A 0.015,B 0.000,C -180.000} C_DIS
LIN {X -219.126,Y 267.875,Z -30.000,A 0.015,B -0.000,C 180.000} C_DIS
LIN {X -218.945,Y 267.847,Z -30.000,A 0.015,B 0.000,C 180.000} C_DIS
LIN {X -215.317,Y 267.391,Z -30.000,A 0.015,B 0.000,C 180.000} C_DIS
LIN {X -214.895,Y 267.364,Z -30.000,A 0.015,B 0.000,C 180.000} C_DIS
LIN {X -178.617,Y 267.364,Z -30.000,A 0.015,B -0.000,C -180.000} C_DIS
LIN {X -178.195,Y 267.391,Z -30.000,A 0.015,B 0.000,C 180.000} C_DIS
LIN {X -174.567,Y 267.847,Z -30.000,A 0.015,B 0.000,C -180.000} C_DIS
LIN {X -174.386,Y 267.875,Z -30.000,A 0.015,B 0.000,C 180.000} C_DIS
LIN {X -170.033,Y 268.663,Z -30.000,A 0.015,B 0.000,C -180.000} C_DIS
LIN {X -169.587,Y 268.775,Z -30.000,A 0.015,B 0.000,C 180.000} C_DIS
LIN {X -167.474,Y 269.464,Z -30.000,A 0.015,B -0.000,C -180.000} C_DIS
LIN {X -167.118,Y 269.603,Z -30.000,A 0.015,B 0.000,C 180.000} C_DIS
LIN {X -164.877,Y 270.626,Z -30.000,A 0.015,B 0.000,C 180.000} C_DIS
LIN {X -164.495,Y 270.831,Z -30.000,A 0.015,B 0.000,C -180.000} C_DIS
LIN {X -161.593,Y 272.636,Z -30.000,A 0.015,B 0.000,C 180.000} C_DIS
LIN {X -161.361,Y 272.794,Z -30.000,A 0.015,B 0.000,C 180.000} C_DIS
LIN {X -157.000,Y 276.038,Z -30.000,A 0.015,B 0.000,C 180.000} C_DIS
LIN {X -156.450,Y 276.551,Z -30.000,A 0.015,B 0.000,C 180.000} C_DIS
LIN {X -154.487,Y 278.844,Z -30.000,A 0.015,B -0.000,C 180.000} C_DIS
LIN {X -154.322,Y 279.052,Z -30.000,A 0.015,B 0.000,C 180.000} C_DIS
LIN {X -151.939,Y 282.321,Z -30.000,A 0.015,B 0.000,C -180.000} C_DIS
LIN {X -151.715,Y 282.673,Z -30.000,A 0.015,B -0.000,C 180.000} C_DIS
LIN {X -149.770,Y 286.181,Z -30.000,A 0.015,B 0.000,C 180.000} C_DIS
LIN {X -149.437,Y 287.041,Z -30.000,A 0.015,B 0.000,C -180.000} C_DIS
LIN {X -147.117,Y 296.835,Z -30.000,A 0.015,B 0.000,C 180.000} C_DIS
LIN {X -147.029,Y 297.453,Z -30.000,A 0.015,B 0.000,C -180.000} C_DIS
LIN {X -146.995,Y 298.179,Z -30.000,A 0.015,B 0.000,C 180.000} C_DIS
LIN {X -147.027,Y 298.837,Z -30.000,A 0.015,B 0.000,C 180.000} C_DIS
LIN {X -148.481,Y 308.631,Z -30.000,A 0.015,B 0.000,C -180.000} C_DIS
LIN {X -148.635,Y 309.254,Z -30.000,A 0.015,B 0.000,C -180.000} C_DIS
LIN {X -149.271,Y 311.067,Z -30.000,A 0.015,B 0.000,C -180.000} C_DIS
LIN {X -149.482,Y 311.547,Z -30.000,A 0.015,B -0.000,C -180.000} C_DIS
LIN {X -151.428,Y 315.175,Z -30.000,A 0.015,B 0.000,C 180.000} C_DIS
LIN {X -151.458,Y 315.229,Z -30.000,A 0.015,B -0.000,C -180.000} C_DIS
LIN {X -155.119,Y 321.759,Z -30.000,A 0.015,B -0.000,C 180.000} C_DIS
LIN {X -155.444,Y 322.237,Z -30.000,A 0.015,B 0.000,C 180.000} C_DIS
LIN {X -156.622,Y 323.688,Z -30.000,A 0.015,B 0.000,C -180.000} C_DIS
LIN {X -156.916,Y 324.006,Z -30.000,A 0.015,B -0.000,C -180.000} C_DIS
LIN {X -165.038,Y 331.737,Z -30.000,A 0.015,B 0.000,C -180.000} C_DIS
LIN {X -165.336,Y 331.990,Z -30.000,A 0.015,B -0.000,C -180.000} C_DIS
LIN {X -166.425,Y 332.809,Z -30.000,A 0.015,B 0.000,C 180.000} C_DIS
LIN {X -166.966,Y 333.142,Z -30.000,A 0.015,B 0.000,C -180.000} C_DIS
LIN {X -177.850,Y 338.493,Z -30.000,A 0.015,B 0.000,C -180.000} C_DIS
LIN {X -178.188,Y 338.637,Z -30.000,A 0.015,B 0.000,C 180.000} C_DIS
LIN {X -178.913,Y 338.900,Z -30.000,A 0.015,B 0.000,C -180.000} C_DIS
LIN {X -179.550,Y 339.063,Z -30.000,A 0.015,B 0.000,C 180.000} C_DIS
LIN {X -180.459,Y 339.204,Z -30.000,A 0.015,B 0.000,C 180.000} C_DIS
LIN {X 4.865,Y 339.209,Z -30.000,A 0.015,B 0.000,C -180.000} C_DIS
LIN {X 5.937,Y 339.152,Z -30.000,A 0.015,B 0.000,C 180.000} C_DIS
LIN {X 6.802,Y 338.955,Z -30.000,A 0.015,B 0.000,C 180.000} C_DIS
LIN {X 7.069,Y 338.840,Z -30.000,A 0.015,B 0.000,C -180.000} C_DIS
LIN {X 7.374,Y 338.634,Z -30.000,A 0.015,B -0.000,C -180.000} C_DIS
LIN {X 9.664,Y 336.377,Z -30.000,A 0.015,B 0.000,C 180.000} C_DIS
LIN {X 9.898,Y 336.018,Z -30.000,A 0.015,B 0.000,C 180.000} C_DIS
LIN {X 10.072,Y 335.556,Z -30.000,A 0.015,B -0.000,C 180.000} C_DIS
LIN {X 10.265,Y 334.347,Z -30.000,A 0.015,B 0.000,C 180.000} C_DIS
LIN {X 10.273,Y 31.844,Z -30.000,A 0.015,B -0.000,C -180.000} C_DIS
LIN {X 9.143,Y 36.475,Z -30.000,A 0.015,B 0.000,C 180.000} C_DIS
LIN {X 9.023,Y 36.864,Z -30.000,A 0.015,B 0.000,C -180.000} C_DIS
LIN {X 8.506,Y 38.240,Z -30.000,A 0.015,B -0.000,C -180.000} C_DIS
LIN {X 8.269,Y 38.741,Z -30.000,A 0.015,B 0.000,C 180.000} C_DIS
LIN {X 6.110,Y 42.480,Z -30.000,A 0.015,B -0.000,C 180.000} C_DIS
LIN {X 6.063,Y 42.560,Z -30.000,A 0.015,B -0.000,C -180.000} C_DIS
LIN {X 2.274,Y 48.726,Z -30.000,A 0.015,B -0.000,C -180.000} C_DIS
LIN {X 2.069,Y 49.024,Z -30.000,A 0.015,B -0.000,C -180.000} C_DIS
LIN {X 1.041,Y 50.353,Z -30.000,A 0.015,B 0.000,C 180.000} C_DIS
LIN {X 0.485,Y 50.920,Z -30.000,A 0.015,B -0.000,C 180.000} C_DIS
LIN {X -7.437,Y 57.295,Z -30.000,A 0.015,B 0.000,C -180.000} C_DIS
LIN {X -7.811,Y 57.556,Z -30.000,A 0.015,B 0.000,C 180.000} C_DIS
LIN {X -8.477,Y 57.958,Z -30.000,A 0.015,B -0.000,C -180.000} C_DIS
LIN {X -9.247,Y 58.300,Z -30.000,A 0.015,B -0.000,C 180.000} C_DIS
LIN {X -19.101,Y 61.273,Z -30.000,A 0.015,B 0.000,C -180.000} C_DIS
LIN {X -19.996,Y 61.416,Z -30.000,A 0.015,B 0.000,C 180.000} C_DIS
LIN {X -23.261,Y 61.496,Z -30.000,A 0.015,B 0.000,C 180.000} C_DIS
LIN {X -23.603,Y 61.487,Z -30.000,A 0.015,B 0.000,C 180.000} C_DIS
LIN {X -27.231,Y 61.207,Z -30.000,A 0.015,B -0.000,C 180.000} C_DIS
LIN {X -27.550,Y 61.167,Z -30.000,A 0.015,B 0.000,C 180.000} C_DIS
LIN {X -31.540,Y 60.474,Z -30.000,A 0.015,B 0.000,C 180.000} C_DIS
LIN {X -32.268,Y 60.261,Z -30.000,A 0.015,B 0.000,C -180.000} C_DIS
LIN {X -36.668,Y 58.419,Z -30.000,A 0.015,B 0.000,C 180.000} C_DIS
LIN {X -36.894,Y 58.314,Z -30.000,A 0.015,B 0.000,C 180.000} C_DIS
LIN {X -40.112,Y 56.679,Z -30.000,A 0.015,B 0.000,C 180.000} C_DIS
LIN {X -40.472,Y 56.467,Z -30.000,A 0.015,B 0.000,C -180.000} C_DIS
LIN {X -42.349,Y 55.201,Z -30.000,A 0.015,B 0.000,C -180.000} C_DIS
LIN {X -42.658,Y 54.965,Z -30.000,A 0.015,B 0.000,C 180.000} C_DIS
LIN {X -44.717,Y 53.201,Z -30.000,A 0.015,B 0.000,C 180.000} C_DIS
LIN {X -45.043,Y 52.881,Z -30.000,A 0.015,B 0.000,C 180.000} C_DIS
LIN {X -46.912,Y 50.781,Z -30.000,A 0.015,B 0.000,C -180.000} C_DIS
LIN {X -47.053,Y 50.612,Z -30.000,A 0.015,B -0.000,C -180.000} C_DIS
LIN {X -50.384,Y 46.336,Z -30.000,A 0.015,B 0.000,C 180.000} C_DIS
LIN {X -50.645,Y 45.950,Z -30.000,A 0.015,B 0.000,C -180.000} C_DIS
LIN {X -68.791,Y 14.550,Z -30.000,A 0.015,B 0.000,C 180.000} C_DIS
LIN {X -68.976,Y 14.178,Z -30.000,A 0.015,B 0.000,C 180.000} C_DIS
LIN {X -70.669,Y 10.188,Z -30.000,A 0.015,B 0.000,C -180.000} C_DIS
LIN {X -70.746,Y 9.989,Z -30.000,A 0.015,B 0.000,C -180.000} C_DIS
LIN {X -72.021,Y 6.362,Z -30.000,A 0.015,B -0.000,C 180.000} C_DIS
LIN {X -72.138,Y 5.945,Z -30.000,A 0.015,B 0.000,C -180.000} C_DIS
LIN {X -72.602,Y 3.768,Z -30.000,A 0.015,B 0.000,C 180.000} C_DIS
LIN {X -72.662,Y 3.377,Z -30.000,A 0.015,B 0.000,C 180.000} C_DIS
LIN {X -72.932,Y 0.475,Z -30.000,A 0.015,B 0.000,C -180.000} C_DIS
LIN {X -72.943,Y 0.005,Z -30.000,A 0.015,B -0.000,C 180.000} C_DIS
LIN {X -72.809,Y -2.897,Z -30.000,A 0.015,B 0.000,C -180.000} C_DIS
LIN {X -72.791,Y -3.122,Z -30.000,A 0.015,B 0.000,C -180.000} C_DIS
LIN {X -72.174,Y -8.563,Z -30.000,A 0.015,B 0.000,C 180.000} C_DIS
LIN {X -72.004,Y -9.304,Z -30.000,A 0.015,B 0.000,C 180.000} C_DIS
LIN {X -70.794,Y -12.744,Z -30.000,A 0.015,B 0.000,C 180.000} C_DIS
LIN {X -70.679,Y -13.029,Z -30.000,A 0.015,B 0.000,C -180.000} C_DIS
LIN {X -69.264,Y -16.119,Z -30.000,A 0.015,B 0.000,C 180.000} C_DIS
LIN {X -69.119,Y -16.400,Z -30.000,A 0.015,B 0.000,C 180.000} C_DIS
LIN {X -67.656,Y -18.939,Z -30.000,A 0.015,B 0.000,C 180.000} C_DIS
LIN {X -67.524,Y -19.150,Z -30.000,A 0.015,B 0.000,C 180.000} C_DIS
LIN {X -66.768,Y -20.264,Z -30.000,A 0.015,B 0.000,C -180.000} C_DIS
LIN {X -66.289,Y -20.826,Z -30.000,A 0.015,B 0.000,C -180.000} C_DIS
LIN {X -59.765,Y -26.973,Z -30.000,A 0.015,B 0.000,C 180.000} C_DIS
LIN {X -59.605,Y -27.114,Z -30.000,A 0.015,B 0.000,C 180.000} C_DIS
LIN {X -58.517,Y -28.017,Z -30.000,A 0.015,B -0.000,C 180.000} C_DIS
CIRC {X -58.084,Y -28.323,Z -30.000,A 0.015,B 0.000,C 180.000},{X -57.609,Y -28.557,Z -30.000,A 0.015,B 0.000,C -180.000} C_DIS
LIN {X -50.808,Y -31.266,Z -30.000,A 0.015,B 0.000,C 180.000} C_DIS
LIN {X -342.732,Y -31.266,Z -30.000,A 0.015,B 0.000,C -180.000} C_DIS
LIN {X -336.289,Y -28.753,Z -30.000,A 0.015,B 0.000,C 180.000} C_DIS
LIN {X -335.785,Y -28.507,Z -30.000,A 0.015,B -0.000,C 180.000} C_DIS
LIN {X -335.059,Y -28.074,Z -30.000,A 0.015,B -0.000,C 180.000} C_DIS
LIN {X -334.481,Y -27.638,Z -30.000,A 0.015,B -0.000,C 180.000} C_DIS
LIN {X -327.594,Y -21.191,Z -30.000,A 0.015,B 0.000,C 180.000} C_DIS
LIN {X -327.400,Y -20.993,Z -30.000,A 0.015,B 0.000,C 180.000} C_DIS
LIN {X -326.752,Y -20.278,Z -30.000,A 0.015,B 0.000,C -180.000} C_DIS
LIN {X -326.355,Y -19.742,Z -30.000,A 0.015,B -0.000,C 180.000} C_DIS
LIN {X -324.602,Y -16.809,Z -30.000,A 0.015,B 0.000,C 180.000} C_DIS
LIN {X -324.436,Y -16.494,Z -30.000,A 0.015,B -0.000,C 180.000} C_DIS
LIN {X -322.839,Y -13.041,Z -30.000,A 0.015,B 0.000,C 180.000} C_DIS
LIN {X -322.718,Y -12.744,Z -30.000,A 0.015,B 0.000,C 180.000} C_DIS
LIN {X -321.508,Y -9.304,Z -30.000,A 0.015,B -0.000,C 180.000} C_DIS
LIN {X -321.338,Y -8.563,Z -30.000,A 0.015,B 0.000,C 180.000} C_DIS
LIN {X -320.721,Y -3.122,Z -30.000,A 0.015,B 0.000,C 180.000} C_DIS
LIN {X -320.703,Y -2.897,Z -30.000,A 0.015,B 0.000,C -180.000} C_DIS
LIN {X -320.569,Y 0.005,Z -30.000,A 0.015,B 0.000,C 180.000} C_DIS
LIN {X -320.575,Y 0.416,Z -30.000,A 0.015,B -0.000,C 180.000} C_DIS
LIN {X -320.740,Y 2.593,Z -30.000,A 0.015,B 0.000,C -180.000} C_DIS
LIN {X -320.793,Y 2.989,Z -30.000,A 0.015,B -0.000,C 180.000} C_DIS
LIN {X -321.363,Y 5.891,Z -30.000,A 0.015,B -0.000,C 180.000} C_DIS
LIN {X -321.489,Y 6.356,Z -30.000,A 0.015,B 0.000,C -180.000} C_DIS
LIN {X -322.716,Y 9.868,Z -30.000,A 0.015,B 0.000,C -180.000} C_DIS
LIN {X -322.788,Y 10.057,Z -30.000,A 0.015,B 0.000,C 180.000} C_DIS
LIN {X -324.354,Y 13.800,Z -30.000,A 0.015,B 0.000,C 180.000} C_DIS
LIN {X -324.544,Y 14.184,Z -30.000,A 0.015,B 0.000,C -180.000} C_DIS
LIN {X -342.684,Y 45.663,Z -30.000,A 0.015,B -0.000,C -180.000} C_DIS
LIN {X -342.906,Y 46.000,Z -30.000,A 0.015,B 0.000,C -180.000} C_DIS
LIN {X -344.864,Y 48.619,Z -30.000,A 0.015,B 0.000,C -180.000} C_DIS
LIN {X -344.971,Y 48.754,Z -30.000,A 0.015,B -0.000,C 180.000} C_DIS
LIN {X -347.854,Y 52.225,Z -30.000,A 0.015,B 0.000,C 180.000} C_DIS
LIN {X -348.147,Y 52.536,Z -30.000,A 0.015,B -0.000,C 180.000} C_DIS
LIN {X -350.233,Y 54.484,Z -30.000,A 0.015,B 0.000,C 180.000} C_DIS
LIN {X -350.597,Y 54.780,Z -30.000,A 0.015,B 0.000,C 180.000} C_DIS
LIN {X -352.518,Y 56.130,Z -30.000,A 0.015,B -0.000,C 180.000} C_DIS
LIN {X -352.875,Y 56.349,Z -30.000,A 0.015,B 0.000,C 180.000} C_DIS
LIN {X -356.247,Y 58.141,Z -30.000,A 0.015,B 0.000,C 180.000} C_DIS
LIN {X -356.489,Y 58.257,Z -30.000,A 0.015,B 0.000,C -180.000} C_DIS
LIN {X -360.843,Y 60.144,Z -30.000,A 0.015,B 0.000,C 180.000} C_DIS
LIN {X -361.542,Y 60.360,Z -30.000,A 0.015,B 0.000,C -180.000} C_DIS
LIN {X -365.170,Y 61.066,Z -30.000,A 0.015,B 0.000,C 180.000} C_DIS
LIN {X -365.485,Y 61.112,Z -30.000,A 0.015,B 0.000,C 180.000} C_DIS
LIN {X -369.113,Y 61.468,Z -30.000,A 0.015,B 0.000,C -180.000} C_DIS
LIN {X -369.500,Y 61.484,Z -30.000,A 0.015,B 0.000,C 180.000} C_DIS
LIN {X -373.490,Y 61.417,Z -30.000,A 0.015,B 0.000,C 180.000} C_DIS
LIN {X -374.399,Y 61.277,Z -30.000,A 0.015,B 0.000,C 180.000} C_DIS
LIN {X -383.587,Y 58.541,Z -30.000,A 0.015,B -0.000,C -180.000} C_DIS
LIN {X -383.914,Y 58.425,Z -30.000,A 0.015,B 0.000,C 180.000} C_DIS
LIN {X -384.914,Y 58.011,Z -30.000,A 0.015,B 0.000,C -180.000} C_DIS
LIN {X -385.721,Y 57.538,Z -30.000,A 0.015,B -0.000,C 180.000} C_DIS
LIN {X -393.652,Y 51.260,Z -30.000,A 0.015,B 0.000,C 180.000} C_DIS
LIN {X -394.117,Y 50.812,Z -30.000,A 0.015,B -0.000,C 180.000} C_DIS
LIN {X -395.226,Y 49.522,Z -30.000,A 0.015,B 0.000,C -180.000} C_DIS
LIN {X -395.532,Y 49.106,Z -30.000,A 0.015,B 0.000,C -180.000} C_DIS
LIN {X -397.792,Y 45.480,Z -30.000,A 0.015,B -0.000,C -180.000} C_DIS
LIN {X -397.832,Y 45.414,Z -30.000,A 0.015,B 0.000,C 180.000} C_DIS
LIN {X -401.763,Y 38.772,Z -30.000,A 0.015,B 0.000,C -180.000} C_DIS
LIN {X -401.989,Y 38.314,Z -30.000,A 0.015,B 0.000,C 180.000} C_DIS
LIN {X -402.405,Y 37.281,Z -30.000,A 0.015,B 0.000,C -180.000} C_DIS
LIN {X -402.546,Y 36.852,Z -30.000,A 0.015,B -0.000,C 180.000} C_DIS
LIN {X -403.548,Y 32.918,Z -30.000,A 0.015,B -0.000,C 180.000} C_DIS
LIN {X -403.561,Y 32.864,Z -30.000,A 0.015,B -0.000,C 180.000} C_DIS
LIN {X -403.779,Y 31.947,Z -30.000,A 0.015,B -0.000,C -180.000} C_DIS
LIN {X -403.787,Y 333.800,Z -30.000,A 0.015,B -0.000,C 180.000} C_DIS
LIN {X -403.730,Y 334.871,Z -30.000,A 0.015,B 0.000,C -180.000} C_DIS
LIN {X -403.533,Y 335.736,Z -30.000,A 0.015,B -0.000,C -180.000} C_DIS
LIN {X -403.418,Y 336.003,Z -30.000,A 0.015,B 0.000,C 180.000} C_DIS
LIN {X -403.034,Y 336.500,Z -29.830,A 0.015,B -0.000,C -180.000} C_DIS
LIN {X -402.624,Y 336.714,Z -29.365,A 0.015,B -0.000,C -180.000} C_DIS
LIN {X -402.458,Y 336.753,Z -28.730,A 0.015,B -0.000,C -180.000} C_DIS
$VEL.CP = 1.00000
LIN {X -402.458,Y 336.753,Z 11.000,A 0.015,B 0.000,C 180.000} C_DIS
$VEL.CP = 1.00000
LIN {X -212.830,Y 109.481,Z 11.000,A 0.015,B 0.000,C 180.000} C_DIS
$VEL.CP = 1.00000
LIN {X -212.830,Y 109.481,Z -18.231,A 0.015,B 0.000,C -180.000} C_DIS
$VEL.CP = 0.10000
LIN {X -212.668,Y 109.462,Z -18.853,A 0.015,B -0.000,C -180.000} C_DIS
LIN {X -212.222,Y 109.434,Z -19.316,A 0.015,B 0.000,C 180.000} C_DIS
LIN {X -211.606,Y 109.450,Z -19.500,A 0.015,B 0.000,C 180.000} C_DIS
LIN {X -206.370,Y 113.474,Z -19.744,A 0.015,B 0.000,C 180.000} C_DIS
LIN {X -207.958,Y 119.884,Z -19.988,A 0.015,B -0.000,C 180.000} C_DIS
LIN {X -214.468,Y 120.998,Z -20.232,A 0.015,B 0.000,C 180.000} C_DIS
LIN {X -218.097,Y 115.479,Z -20.476,A 0.015,B -0.000,C -180.000} C_DIS
LIN {X -214.495,Y 109.944,Z -20.720,A 0.015,B 0.000,C 180.000} C_DIS
LIN {X -207.980,Y 111.025,Z -20.964,A 0.015,B 0.000,C -180.000} C_DIS
LIN {X -206.360,Y 117.428,Z -21.208,A 0.015,B 0.000,C 180.000} C_DIS
LIN {X -211.577,Y 121.477,Z -21.452,A 0.015,B 0.000,C 180.000} C_DIS
LIN {X -217.378,Y 118.321,Z -21.696,A 0.015,B 0.000,C 180.000} C_DIS
LIN {X -216.810,Y 111.741,Z -21.940,A 0.015,B 0.000,C -180.000} C_DIS
LIN {X -210.554,Y 109.624,Z -22.185,A 0.015,B 0.000,C -180.000} C_DIS
LIN {X -206.108,Y 114.508,Z -22.429,A 0.015,B 0.000,C -180.000} C_DIS
LIN {X -208.801,Y 120.538,Z -22.673,A 0.015,B 0.000,C 180.000} C_DIS
LIN {X -215.405,Y 120.488,Z -22.917,A 0.015,B 0.000,C 180.000} C_DIS
LIN {X -218.005,Y 114.417,Z -23.161,A 0.015,B 0.000,C -180.000} C_DIS
LIN {X -213.485,Y 109.602,Z -23.405,A 0.015,B 0.000,C 180.000} C_DIS
LIN {X -207.262,Y 111.814,Z -23.649,A 0.015,B 0.000,C -180.000} C_DIS
LIN {X -206.795,Y 118.402,Z -23.893,A 0.015,B 0.000,C -180.000} C_DIS
LIN {X -212.643,Y 121.469,Z -24.137,A 0.015,B -0.000,C 180.000} C_DIS
LIN {X -217.798,Y 117.340,Z -24.381,A 0.015,B -0.000,C -180.000} C_DIS
LIN {X -216.080,Y 110.963,Z -24.625,A 0.015,B 0.000,C -180.000} C_DIS
LIN {X -209.549,Y 109.981,Z -24.869,A 0.015,B -0.000,C 180.000} C_DIS
LIN {X -206.033,Y 115.572,Z -25.113,A 0.015,B 0.000,C 180.000} C_DIS
LIN {X -209.745,Y 121.034,Z -25.357,A 0.015,B 0.000,C 180.000} C_DIS
LIN {X -216.237,Y 119.821,Z -25.601,A 0.015,B -0.000,C -180.000} C_DIS
LIN {X -217.728,Y 113.387,Z -25.845,A 0.015,B -0.000,C 180.000} C_DIS
LIN {X -212.430,Y 109.443,Z -26.089,A 0.015,B 0.000,C 180.000} C_DIS
LIN {X -206.694,Y 112.717,Z -26.333,A 0.015,B 0.000,C -180.000} C_DIS
LIN {X -207.395,Y 119.284,Z -26.577,A 0.015,B 0.000,C -180.000} C_DIS
LIN {X -213.692,Y 121.273,Z -26.821,A 0.015,B 0.000,C 180.000} C_DIS
LIN {X -218.038,Y 116.301,Z -27.065,A 0.015,B 0.000,C 180.000} C_DIS
LIN {X -215.224,Y 110.326,Z -27.310,A 0.015,B 0.000,C -180.000} C_DIS
LIN {X -208.623,Y 110.510,Z -27.554,A 0.015,B 0.000,C 180.000} C_DIS
LIN {X -206.146,Y 116.632,Z -27.798,A 0.015,B -0.000,C 180.000} C_DIS
LIN {X -210.762,Y 121.355,Z -28.042,A 0.015,B 0.000,C 180.000} C_DIS
LIN {X -216.939,Y 119.018,Z -28.286,A 0.015,B 0.000,C -180.000} C_DIS
LIN {X -217.273,Y 112.422,Z -28.530,A 0.015,B -0.000,C 180.000} C_DIS
LIN {X -211.364,Y 109.473,Z -28.774,A 0.015,B 0.000,C -180.000} C_DIS
LIN {X -206.294,Y 113.705,Z -29.018,A 0.015,B 0.000,C 180.000} C_DIS
LIN {X -208.140,Y 120.046,Z -29.262,A 0.015,B 0.000,C 180.000} C_DIS
